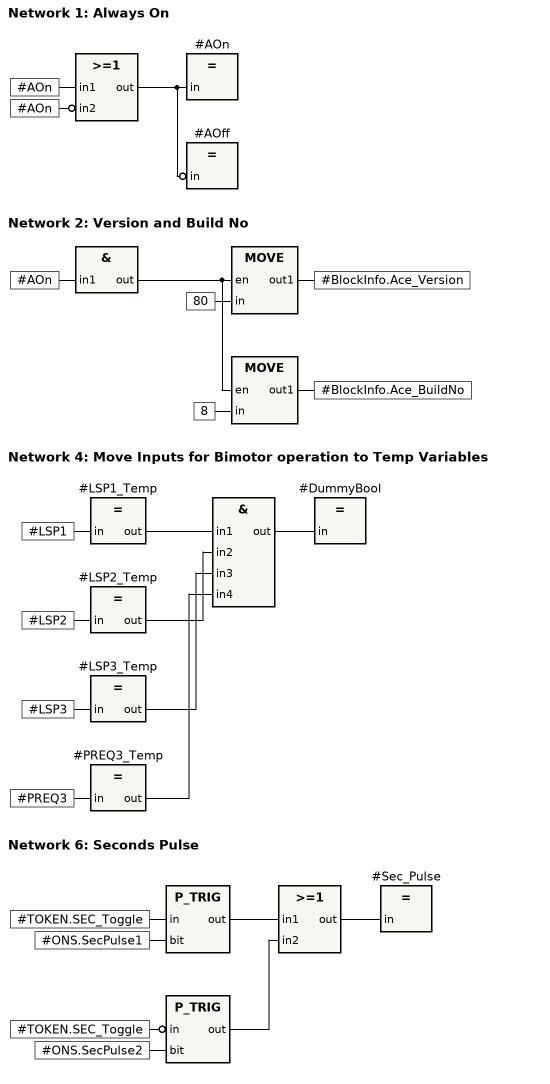
   #AOn := #AOn OR NOT #AOn;
   #AOff := NOT #AOn;
END_REGION

REGION Network 2: Version and Build No
   IF #AOn THEN
       #BlockInfo.Ace_Version := 80;
       #BlockInfo.Ace_BuildNo := 8;
   END_IF;
END_REGION

REGION Network 3 (STL): Instance DB Number to Faceplate
         L     DINO;
         T     #BlockInfo.DB_Number;
END_REGION

REGION Network 4: Move Inputs for Bimotor operation to Temp Variables
   #LSP1_Temp := #LSP1;
   #LSP2_Temp := #LSP2;
   #LSP3_Temp := #LSP3;
   #PREQ3_Temp := #PREQ3;
   #DummyBool := #LSP1 AND #LSP2 AND #LSP3 AND #PREQ3;
END_REGION

REGION Network 5 (SCL): Transfer Interlock OK to Stat
   #OUT.INTL_OK_STAT := PEEK_BOOL(area := 16#84, dbNumber := #BlockInfo.DB_Number, byteOffset := 18, bitOffset := 0);
   #OUT.INTL_SEQ_STR1_OK_STAT := PEEK_BOOL(area := 16#84, dbNumber := #BlockInfo.DB_Number, byteOffset := 20, bitOffset := 0);
   #OUT.INTL_SEQ_STR2_OK_STAT := PEEK_BOOL(area := 16#84, dbNumber := #BlockInfo.DB_Number, byteOffset := 22, bitOffset := 0);
   #OUT.INTL_SEQ_STR3_OK_STAT := PEEK_BOOL(area := 16#84, dbNumber := #BlockInfo.DB_Number, byteOffset := 24, bitOffset := 0);
   #OUT.INTL_SEQ_STP_OK_STAT := PEEK_BOOL(area := 16#84, dbNumber := #BlockInfo.DB_Number, byteOffset := 26, bitOffset := 0);
END_REGION

REGION Network 6: Seconds Pulse
   #_w1 := #TOKEN.SEC_Toggle AND NOT #ONS.SecPulse1;   // rising edge
   #ONS.SecPulse1 := #TOKEN.SEC_Toggle;
   #_w2 := NOT #TOKEN.SEC_Toggle AND NOT #ONS.SecPulse2;   // rising edge
   #ONS.SecPulse2 := NOT #TOKEN.SEC_Toggle;
   #Sec_Pulse := #_w1 OR #_w2;
END_REGION

REGION Network 7: Type Select
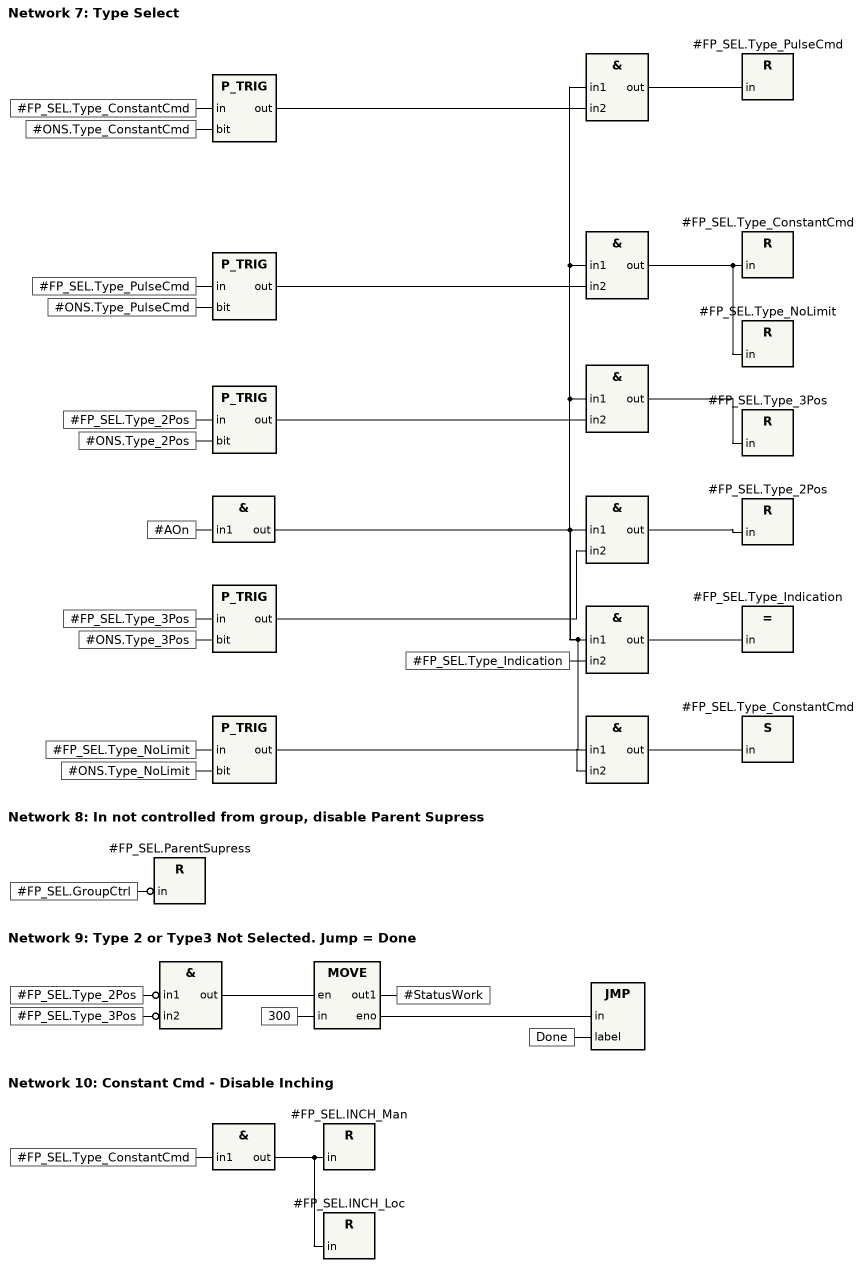
   #_w1 := #FP_SEL.Type_ConstantCmd AND NOT #ONS.Type_ConstantCmd;   // rising edge
   #ONS.Type_ConstantCmd := #FP_SEL.Type_ConstantCmd;
   IF #AOn AND #_w1 THEN #FP_SEL.Type_PulseCmd := FALSE; END_IF;
   #_w2 := #FP_SEL.Type_PulseCmd AND NOT #ONS.Type_PulseCmd;   // rising edge
   #ONS.Type_PulseCmd := #FP_SEL.Type_PulseCmd;
   IF #AOn AND #_w2 THEN
       #FP_SEL.Type_ConstantCmd := FALSE;
       #FP_SEL.Type_NoLimit := FALSE;
   END_IF;
   #_w3 := #FP_SEL.Type_2Pos AND NOT #ONS.Type_2Pos;   // rising edge
   #ONS.Type_2Pos := #FP_SEL.Type_2Pos;
   IF #AOn AND #_w3 THEN #FP_SEL.Type_3Pos := FALSE; END_IF;
   #_w4 := #FP_SEL.Type_3Pos AND NOT #ONS.Type_3Pos;   // rising edge
   #ONS.Type_3Pos := #FP_SEL.Type_3Pos;
   IF #AOn AND #_w4 THEN #FP_SEL.Type_2Pos := FALSE; END_IF;
   #FP_SEL.Type_Indication := #AOn AND #FP_SEL.Type_Indication;
   #_w5 := #FP_SEL.Type_NoLimit AND NOT #ONS.Type_NoLimit;   // rising edge
   #ONS.Type_NoLimit := #FP_SEL.Type_NoLimit;
   IF #AOn AND #_w5 THEN #FP_SEL.Type_ConstantCmd := TRUE; END_IF;
END_REGION

REGION Network 8: In not controlled from group, disable Parent Supress
   IF NOT #FP_SEL.GroupCtrl THEN #FP_SEL.ParentSupress := FALSE; END_IF;
END_REGION

REGION Network 9: Type 2 or Type3 Not Selected. Jump = Done
   // ENO of a box is taken as its EN; it also drops when the box reports an error
   #_w1 := NOT #FP_SEL.Type_2Pos AND NOT #FP_SEL.Type_3Pos;
   IF #_w1 THEN
       #StatusWork := 300;
       GOTO Done;
   END_IF;
END_REGION

REGION Network 10: Constant Cmd - Disable Inching
   IF #FP_SEL.Type_ConstantCmd THEN
       #FP_SEL.INCH_Man := FALSE;
       #FP_SEL.INCH_Loc := FALSE;
   END_IF;
END_REGION

REGION Network 11: Simulate LSP if no limit switches
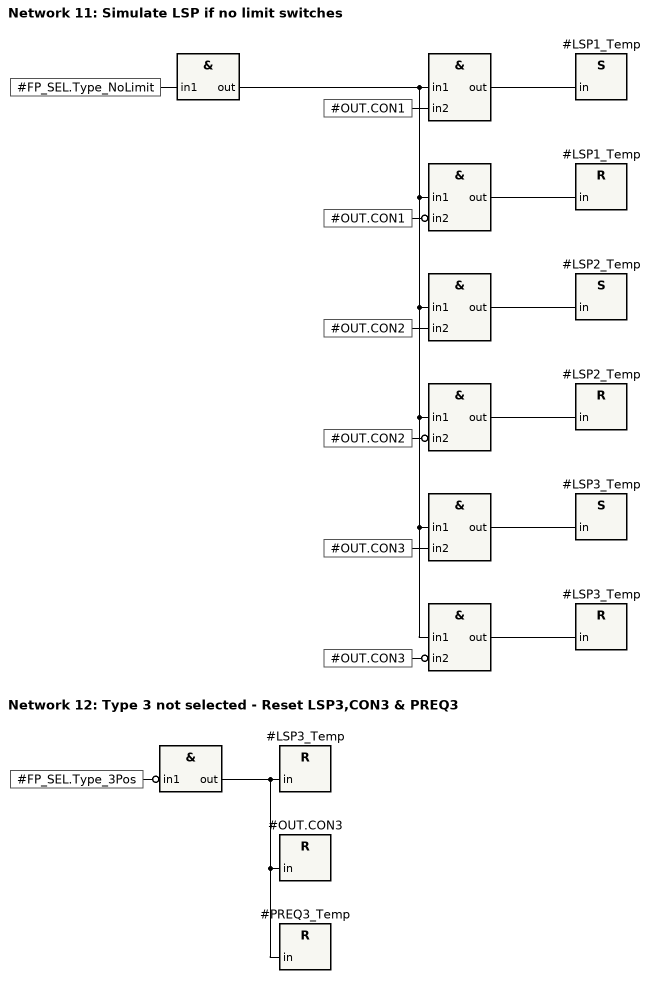
   IF #FP_SEL.Type_NoLimit AND #OUT.CON1 THEN #LSP1_Temp := TRUE; END_IF;
   IF #FP_SEL.Type_NoLimit AND NOT #OUT.CON1 THEN #LSP1_Temp := FALSE; END_IF;
   IF #FP_SEL.Type_NoLimit AND #OUT.CON2 THEN #LSP2_Temp := TRUE; END_IF;
   IF #FP_SEL.Type_NoLimit AND NOT #OUT.CON2 THEN #LSP2_Temp := FALSE; END_IF;
   IF #FP_SEL.Type_NoLimit AND #OUT.CON3 THEN #LSP3_Temp := TRUE; END_IF;
   IF #FP_SEL.Type_NoLimit AND NOT #OUT.CON3 THEN #LSP3_Temp := FALSE; END_IF;
END_REGION

REGION Network 12: Type 3 not selected - Reset LSP3,CON3 & PREQ3
   IF NOT #FP_SEL.Type_3Pos THEN
       #LSP3_Temp := FALSE;
       #OUT.CON3 := FALSE;
       #PREQ3_Temp := FALSE;
   END_IF;
END_REGION

REGION Network 13: Set Show Parameters
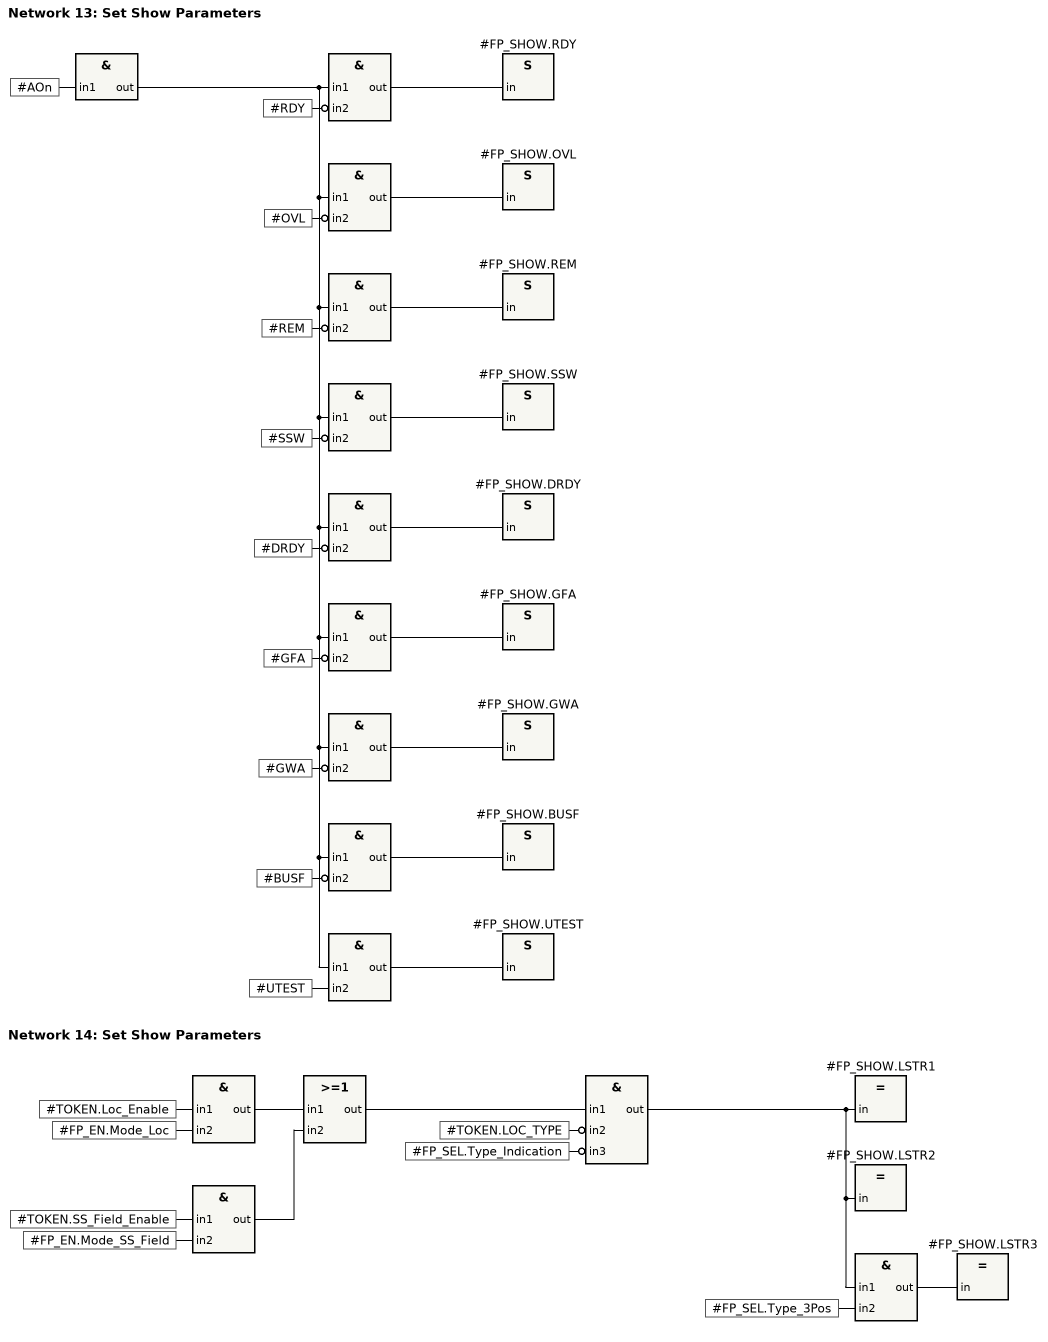
   IF #AOn AND NOT #RDY THEN #FP_SHOW.RDY := TRUE; END_IF;
   IF #AOn AND NOT #OVL THEN #FP_SHOW.OVL := TRUE; END_IF;
   IF #AOn AND NOT #REM THEN #FP_SHOW.REM := TRUE; END_IF;
   IF #AOn AND NOT #SSW THEN #FP_SHOW.SSW := TRUE; END_IF;
   IF #AOn AND NOT #DRDY THEN #FP_SHOW.DRDY := TRUE; END_IF;
   IF #AOn AND NOT #GFA THEN #FP_SHOW.GFA := TRUE; END_IF;
   IF #AOn AND NOT #GWA THEN #FP_SHOW.GWA := TRUE; END_IF;
   IF #AOn AND NOT #BUSF THEN #FP_SHOW.BUSF := TRUE; END_IF;
   IF #AOn AND #UTEST THEN #FP_SHOW.UTEST := TRUE; END_IF;
END_REGION

REGION Network 14: Set Show Parameters
   #FP_SHOW.LSTR1 := ((#TOKEN.Loc_Enable AND #FP_EN.Mode_Loc) OR (#TOKEN.SS_Field_Enable AND #FP_EN.Mode_SS_Field)) AND NOT #TOKEN.LOC_TYPE AND NOT #FP_SEL.Type_Indication;
   #FP_SHOW.LSTR2 := #FP_SHOW.LSTR1;
   #FP_SHOW.LSTR3 := #FP_SHOW.LSTR1 AND #FP_SEL.Type_3Pos;
END_REGION

REGION Network 15: Set Show Parameters
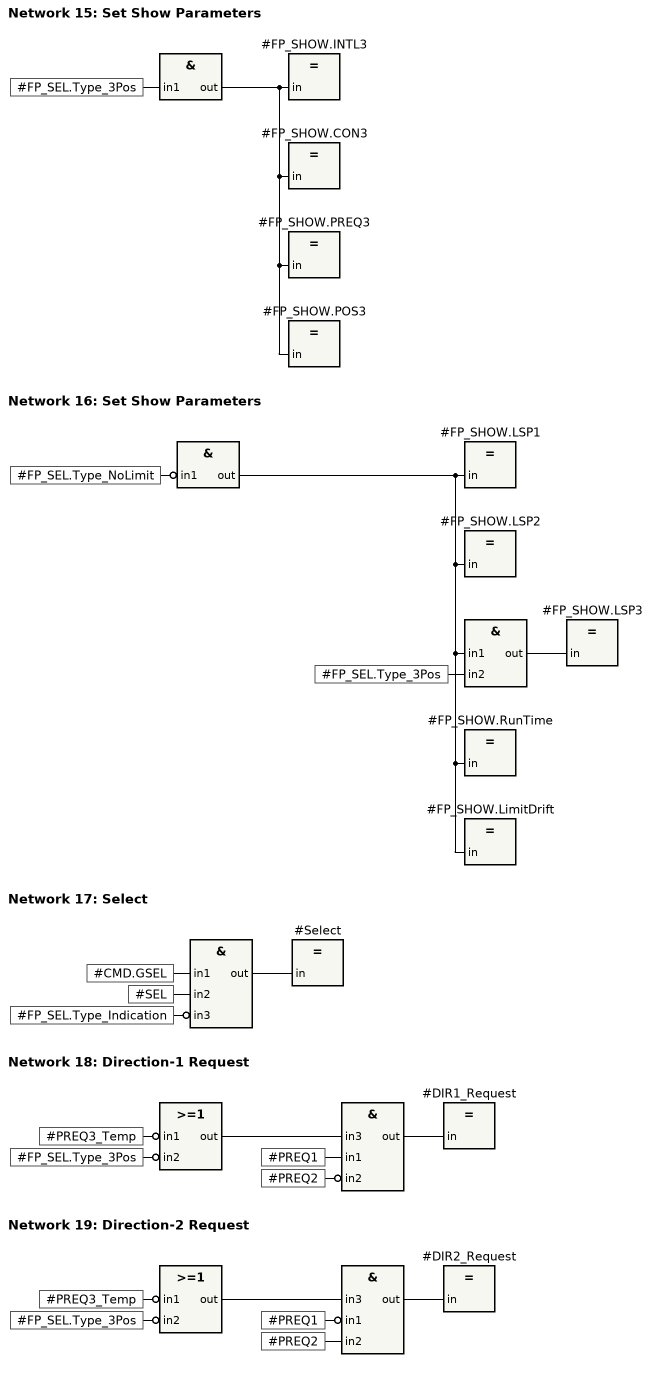
   #FP_SHOW.INTL3 := #FP_SEL.Type_3Pos;
   #FP_SHOW.CON3 := #FP_SEL.Type_3Pos;
   #FP_SHOW.PREQ3 := #FP_SEL.Type_3Pos;
   #FP_SHOW.POS3 := #FP_SEL.Type_3Pos;
END_REGION

REGION Network 16: Set Show Parameters
   #FP_SHOW.LSP1 := NOT #FP_SEL.Type_NoLimit;
   #FP_SHOW.LSP2 := NOT #FP_SEL.Type_NoLimit;
   #FP_SHOW.LSP3 := NOT #FP_SEL.Type_NoLimit AND #FP_SEL.Type_3Pos;
   #FP_SHOW.RunTime := NOT #FP_SEL.Type_NoLimit;
   #FP_SHOW.LimitDrift := NOT #FP_SEL.Type_NoLimit;
END_REGION

REGION Network 17: Select
   #Select := #CMD.GSEL AND #SEL AND NOT #FP_SEL.Type_Indication;
END_REGION

REGION Network 18: Direction-1 Request
   #DIR1_Request := (NOT #PREQ3_Temp OR NOT #FP_SEL.Type_3Pos) AND #PREQ1 AND NOT #PREQ2;
END_REGION

REGION Network 19: Direction-2 Request
   #DIR2_Request := (NOT #PREQ3_Temp OR NOT #FP_SEL.Type_3Pos) AND NOT #PREQ1 AND #PREQ2;
END_REGION

REGION Network 20: Direction-3 Request
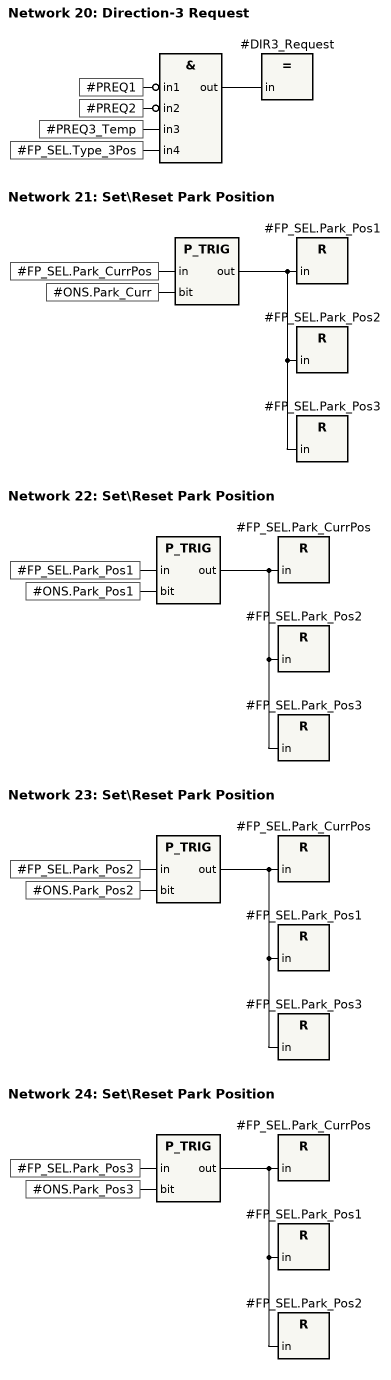
   #DIR3_Request := NOT #PREQ1 AND NOT #PREQ2 AND #PREQ3_Temp AND #FP_SEL.Type_3Pos;
END_REGION

REGION Network 21: Set\Reset Park Position
   #_w1 := #FP_SEL.Park_CurrPos AND NOT #ONS.Park_Curr;   // rising edge
   #ONS.Park_Curr := #FP_SEL.Park_CurrPos;
   IF #_w1 THEN
       #FP_SEL.Park_Pos1 := FALSE;
       #FP_SEL.Park_Pos2 := FALSE;
       #FP_SEL.Park_Pos3 := FALSE;
   END_IF;
END_REGION

REGION Network 22: Set\Reset Park Position
   #_w1 := #FP_SEL.Park_Pos1 AND NOT #ONS.Park_Pos1;   // rising edge
   #ONS.Park_Pos1 := #FP_SEL.Park_Pos1;
   IF #_w1 THEN
       #FP_SEL.Park_CurrPos := FALSE;
       #FP_SEL.Park_Pos2 := FALSE;
       #FP_SEL.Park_Pos3 := FALSE;
   END_IF;
END_REGION

REGION Network 23: Set\Reset Park Position
   #_w1 := #FP_SEL.Park_Pos2 AND NOT #ONS.Park_Pos2;   // rising edge
   #ONS.Park_Pos2 := #FP_SEL.Park_Pos2;
   IF #_w1 THEN
       #FP_SEL.Park_CurrPos := FALSE;
       #FP_SEL.Park_Pos1 := FALSE;
       #FP_SEL.Park_Pos3 := FALSE;
   END_IF;
END_REGION

REGION Network 24: Set\Reset Park Position
   #_w1 := #FP_SEL.Park_Pos3 AND NOT #ONS.Park_Pos3;   // rising edge
   #ONS.Park_Pos3 := #FP_SEL.Park_Pos3;
   IF #_w1 THEN
       #FP_SEL.Park_CurrPos := FALSE;
       #FP_SEL.Park_Pos1 := FALSE;
       #FP_SEL.Park_Pos2 := FALSE;
   END_IF;
END_REGION

REGION Network 25: Set\Reset Park Position
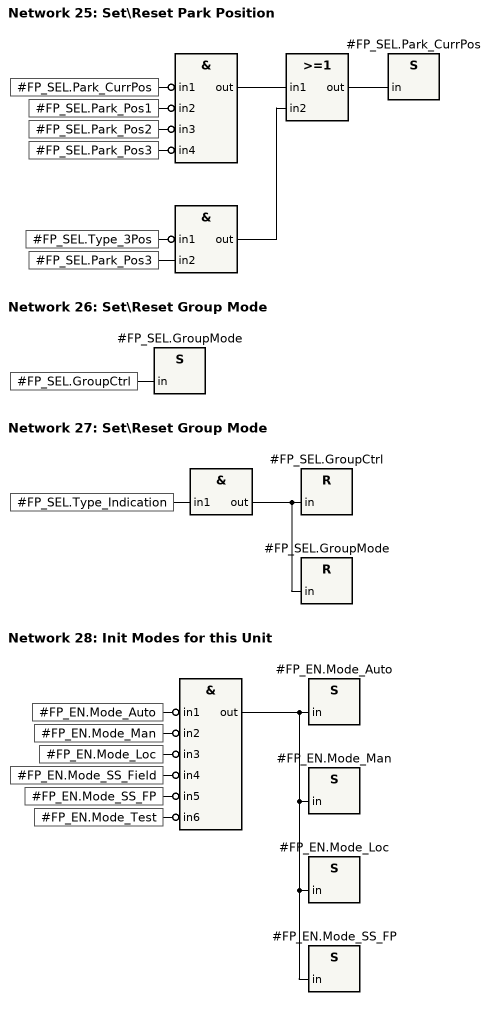
   IF (NOT #FP_SEL.Park_CurrPos AND NOT #FP_SEL.Park_Pos1 AND NOT #FP_SEL.Park_Pos2 AND NOT #FP_SEL.Park_Pos3) OR (NOT #FP_SEL.Type_3Pos AND #FP_SEL.Park_Pos3) THEN
       #FP_SEL.Park_CurrPos := TRUE;
   END_IF;
END_REGION

REGION Network 26: Set\Reset Group Mode
   IF #FP_SEL.GroupCtrl THEN #FP_SEL.GroupMode := TRUE; END_IF;
END_REGION

REGION Network 27: Set\Reset Group Mode
   IF #FP_SEL.Type_Indication THEN
       #FP_SEL.GroupCtrl := FALSE;
       #FP_SEL.GroupMode := FALSE;
   END_IF;
END_REGION

REGION Network 28: Init Modes for this Unit
   #_w1 := NOT #FP_EN.Mode_Auto AND NOT #FP_EN.Mode_Man AND NOT #FP_EN.Mode_Loc AND NOT #FP_EN.Mode_SS_Field AND NOT #FP_EN.Mode_SS_FP AND NOT #FP_EN.Mode_Test;
   IF #_w1 THEN
       #FP_EN.Mode_Auto := TRUE;
       #FP_EN.Mode_Man := TRUE;
       #FP_EN.Mode_Loc := TRUE;
       #FP_EN.Mode_SS_FP := TRUE;
   END_IF;
END_REGION

REGION Network 29: Show Push Buttons on Faceplate
   // build 002 - 27 March 2019 : LOC_Type flag removed from Show_PB_Local
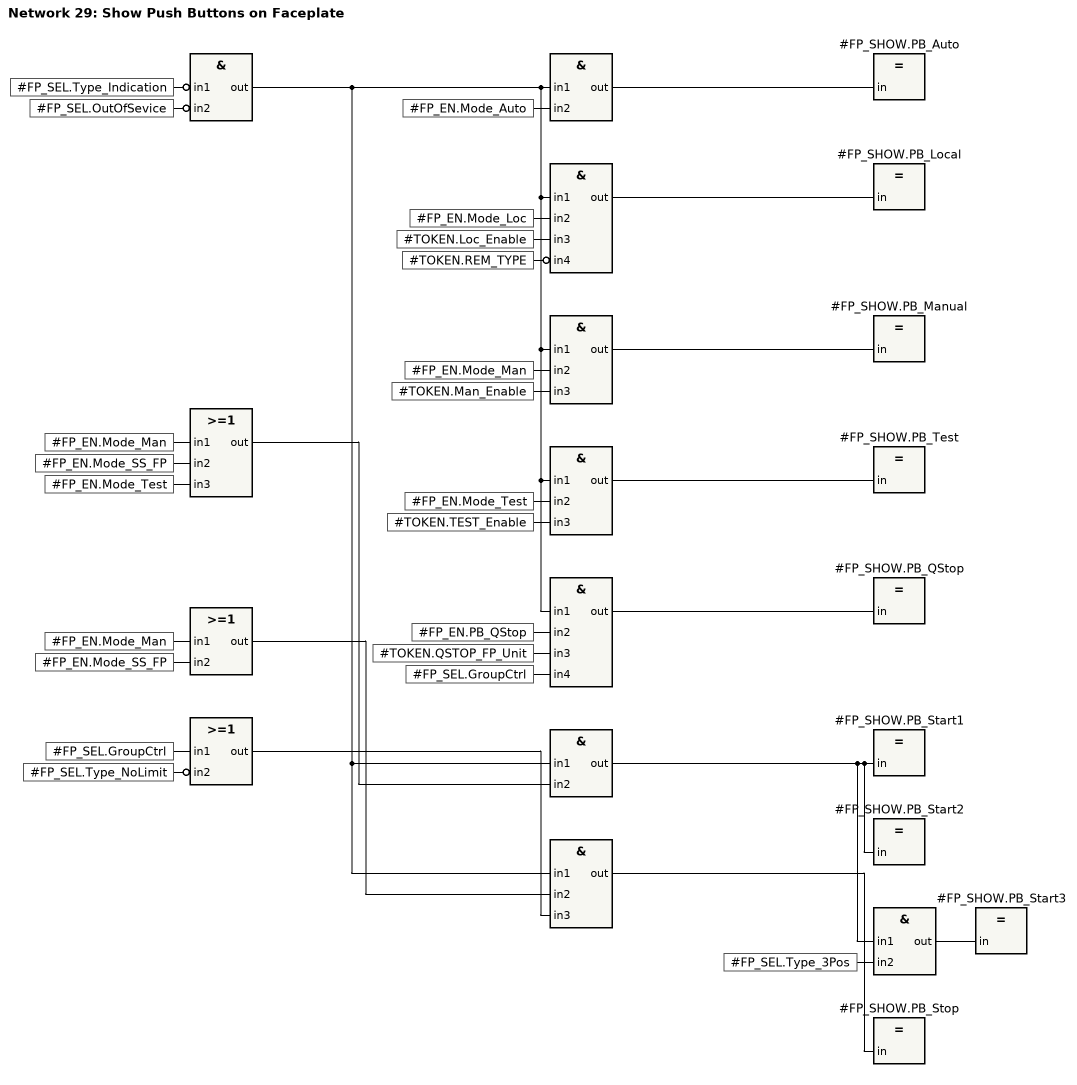
   #_w1 := NOT #FP_SEL.Type_Indication AND NOT #FP_SEL.OutOfSevice;
   #FP_SHOW.PB_Auto := #_w1 AND #FP_EN.Mode_Auto;
   #FP_SHOW.PB_Local := #_w1 AND #FP_EN.Mode_Loc AND #TOKEN.Loc_Enable AND NOT #TOKEN.REM_TYPE;
   #FP_SHOW.PB_Manual := #_w1 AND #FP_EN.Mode_Man AND #TOKEN.Man_Enable;
   #FP_SHOW.PB_Test := #_w1 AND #FP_EN.Mode_Test AND #TOKEN.TEST_Enable;
   #FP_SHOW.PB_QStop := #_w1 AND #FP_EN.PB_QStop AND #TOKEN.QSTOP_FP_Unit AND #FP_SEL.GroupCtrl;
   #FP_SHOW.PB_Start1 := #_w1 AND (#FP_EN.Mode_Man OR #FP_EN.Mode_SS_FP OR #FP_EN.Mode_Test);
   #FP_SHOW.PB_Start2 := #FP_SHOW.PB_Start1;
   #FP_SHOW.PB_Start3 := #FP_SHOW.PB_Start1 AND #FP_SEL.Type_3Pos;
   #FP_SHOW.PB_Stop := #_w1 AND (#FP_EN.Mode_Man OR #FP_EN.Mode_SS_FP) AND (#FP_SEL.GroupCtrl OR NOT #FP_SEL.Type_NoLimit);
END_REGION

REGION Network 30: DimOut Buttons on Faceplate - Auto
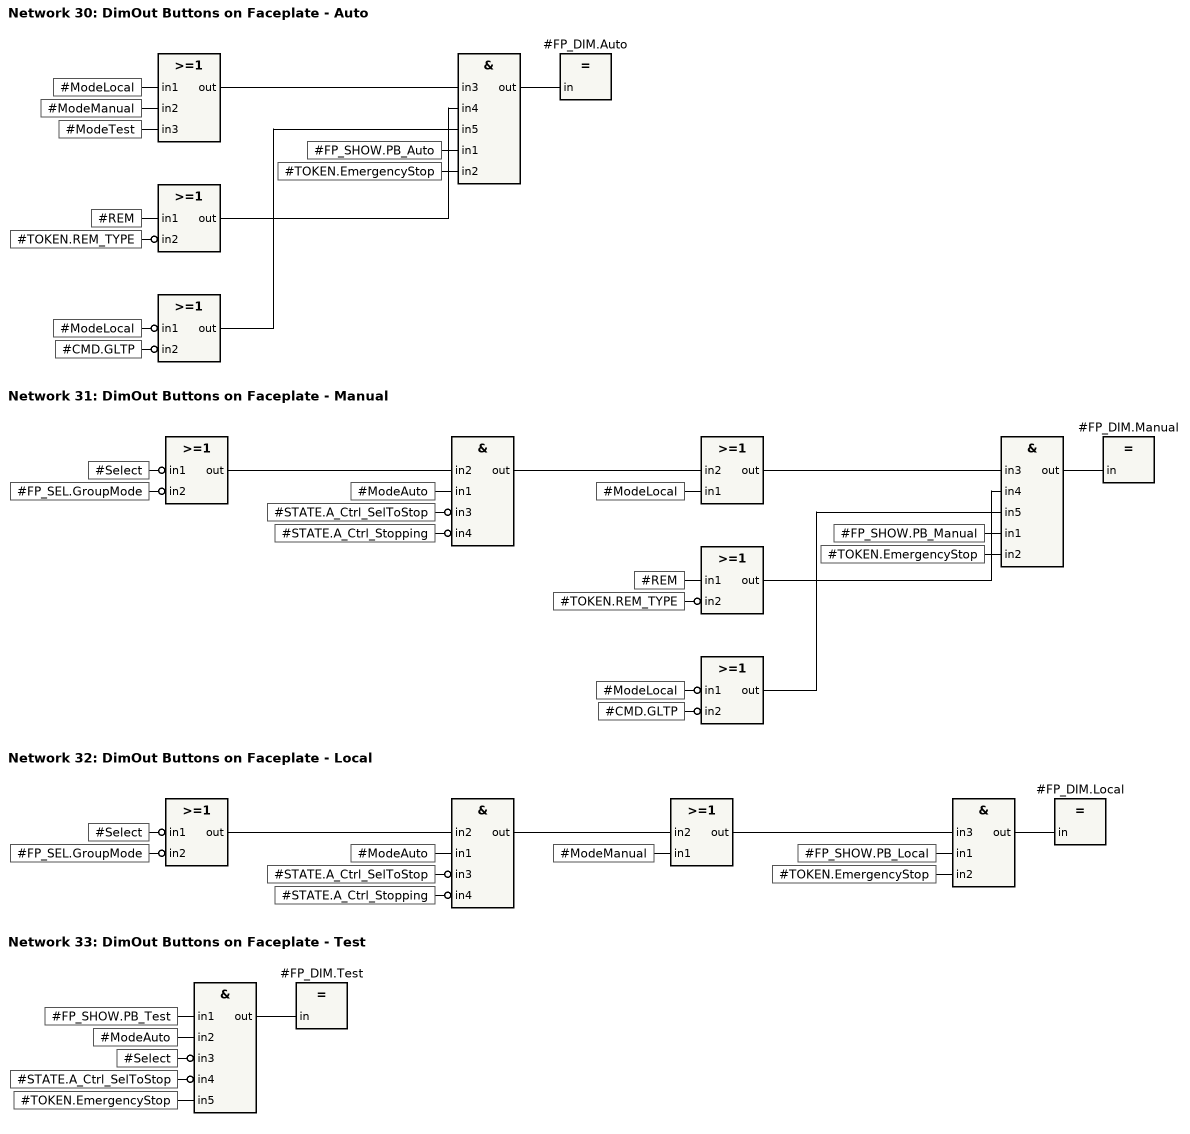
   #FP_DIM.Auto := (#ModeLocal OR #ModeManual OR #ModeTest) AND (#REM OR NOT #TOKEN.REM_TYPE) AND (NOT #ModeLocal OR NOT #CMD.GLTP) AND #FP_SHOW.PB_Auto AND #TOKEN.EmergencyStop;
END_REGION

REGION Network 31: DimOut Buttons on Faceplate - Manual
   #FP_DIM.Manual := (((NOT #Select OR NOT #FP_SEL.GroupMode) AND #ModeAuto AND NOT #STATE.A_Ctrl_SelToStop AND NOT #STATE.A_Ctrl_Stopping) OR #ModeLocal) AND (#REM OR NOT #TOKEN.REM_TYPE) AND (NOT #ModeLocal OR NOT #CMD.GLTP) AND #FP_SHOW.PB_Manual AND #TOKEN.EmergencyStop;
END_REGION

REGION Network 32: DimOut Buttons on Faceplate - Local
   #FP_DIM.Local := (((NOT #Select OR NOT #FP_SEL.GroupMode) AND #ModeAuto AND NOT #STATE.A_Ctrl_SelToStop AND NOT #STATE.A_Ctrl_Stopping) OR #ModeManual) AND #FP_SHOW.PB_Local AND #TOKEN.EmergencyStop;
END_REGION

REGION Network 33: DimOut Buttons on Faceplate - Test
   #FP_DIM.Test := #FP_SHOW.PB_Test AND #ModeAuto AND NOT #Select AND NOT #STATE.A_Ctrl_SelToStop AND #TOKEN.EmergencyStop;
END_REGION

REGION Network 34: DimOut Buttons on Faceplate - Stop
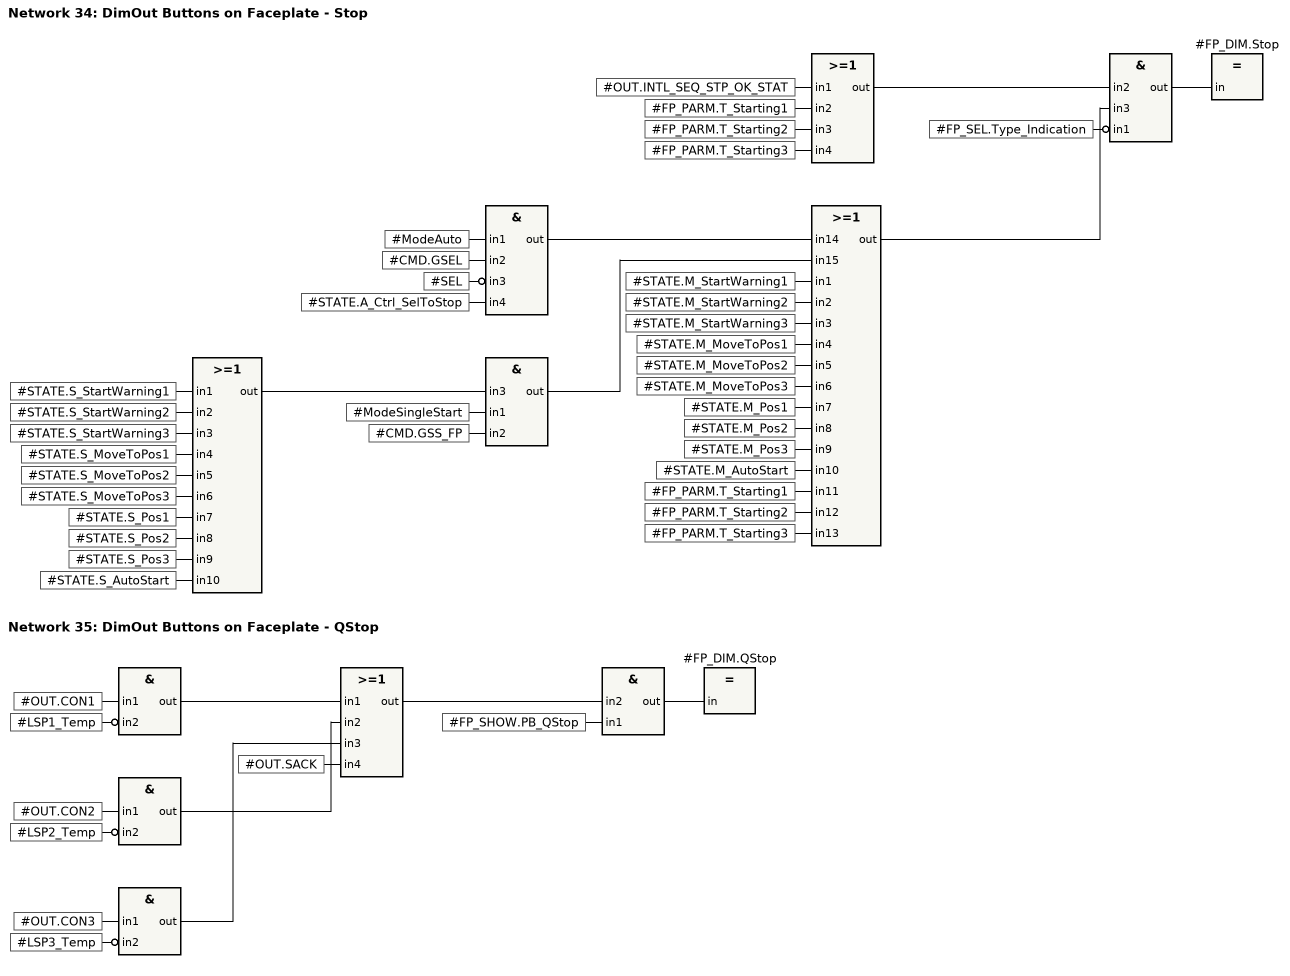
   #FP_DIM.Stop := (#OUT.INTL_SEQ_STP_OK_STAT OR #FP_PARM.T_Starting1 OR #FP_PARM.T_Starting2 OR #FP_PARM.T_Starting3) AND ((#ModeAuto AND #CMD.GSEL AND NOT #SEL AND #STATE.A_Ctrl_SelToStop) OR ((#STATE.S_StartWarning1 OR #STATE.S_StartWarning2 OR #STATE.S_StartWarning3 OR #STATE.S_MoveToPos1 OR #STATE.S_MoveToPos2 OR #STATE.S_MoveToPos3 OR #STATE.S_Pos1 OR #STATE.S_Pos2 OR #STATE.S_Pos3 OR #STATE.S_AutoStart) AND #ModeSingleStart AND #CMD.GSS_FP) OR #STATE.M_StartWarning1 OR #STATE.M_StartWarning2 OR #STATE.M_StartWarning3 OR #STATE.M_MoveToPos1 OR #STATE.M_MoveToPos2 OR #STATE.M_MoveToPos3 OR #STATE.M_Pos1 OR #STATE.M_Pos2 OR #STATE.M_Pos3 OR #STATE.M_AutoStart OR #FP_PARM.T_Starting1 OR #FP_PARM.T_Starting2 OR #FP_PARM.T_Starting3) AND NOT #FP_SEL.Type_Indication;
END_REGION

REGION Network 35: DimOut Buttons on Faceplate - QStop
   #FP_DIM.QStop := ((#OUT.CON1 AND NOT #LSP1_Temp) OR (#OUT.CON2 AND NOT #LSP2_Temp) OR (#OUT.CON3 AND NOT #LSP3_Temp) OR #OUT.SACK) AND #FP_SHOW.PB_QStop;
END_REGION

REGION Network 36: DimOut Buttons on Faceplate - Start1
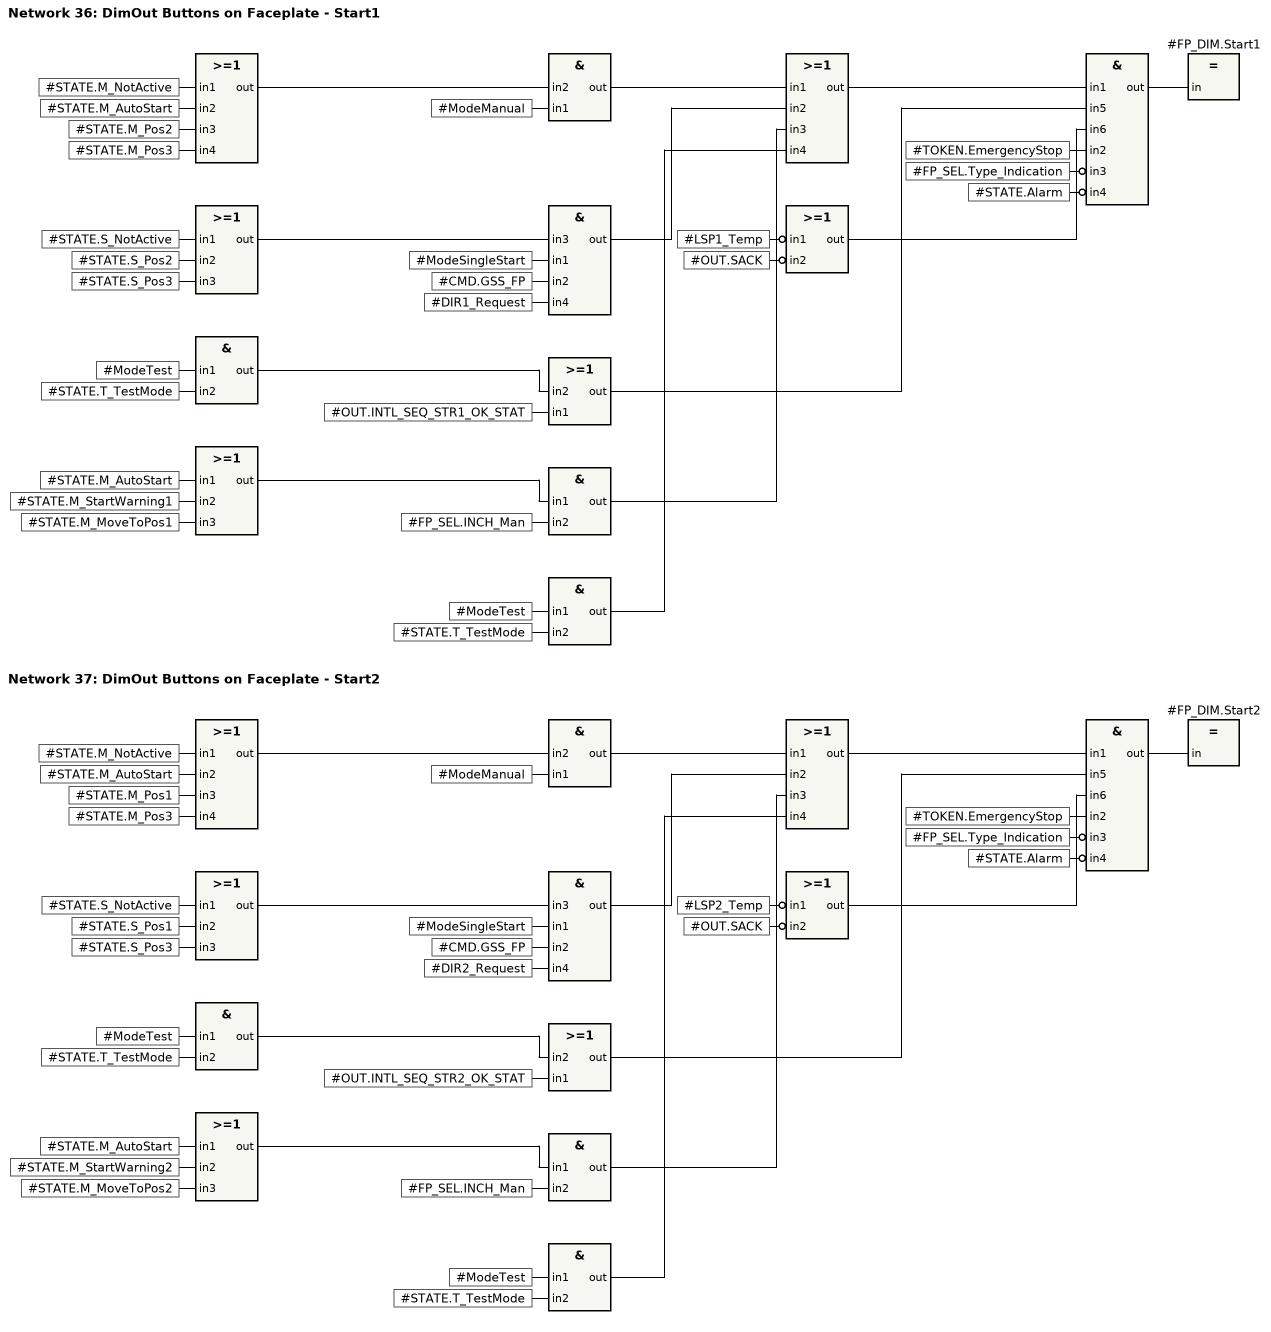
   #FP_DIM.Start1 := (((#STATE.M_NotActive OR #STATE.M_AutoStart OR #STATE.M_Pos2 OR #STATE.M_Pos3) AND #ModeManual) OR ((#STATE.S_NotActive OR #STATE.S_Pos2 OR #STATE.S_Pos3) AND #ModeSingleStart AND #CMD.GSS_FP AND #DIR1_Request) OR ((#STATE.M_AutoStart OR #STATE.M_StartWarning1 OR #STATE.M_MoveToPos1) AND #FP_SEL.INCH_Man) OR (#ModeTest AND #STATE.T_TestMode)) AND ((#ModeTest AND #STATE.T_TestMode) OR #OUT.INTL_SEQ_STR1_OK_STAT) AND (NOT #LSP1_Temp OR NOT #OUT.SACK) AND #TOKEN.EmergencyStop AND NOT #FP_SEL.Type_Indication AND NOT #STATE.Alarm;
END_REGION

REGION Network 37: DimOut Buttons on Faceplate - Start2
   #FP_DIM.Start2 := (((#STATE.M_NotActive OR #STATE.M_AutoStart OR #STATE.M_Pos1 OR #STATE.M_Pos3) AND #ModeManual) OR ((#STATE.S_NotActive OR #STATE.S_Pos1 OR #STATE.S_Pos3) AND #ModeSingleStart AND #CMD.GSS_FP AND #DIR2_Request) OR ((#STATE.M_AutoStart OR #STATE.M_StartWarning2 OR #STATE.M_MoveToPos2) AND #FP_SEL.INCH_Man) OR (#ModeTest AND #STATE.T_TestMode)) AND ((#ModeTest AND #STATE.T_TestMode) OR #OUT.INTL_SEQ_STR2_OK_STAT) AND (NOT #LSP2_Temp OR NOT #OUT.SACK) AND #TOKEN.EmergencyStop AND NOT #FP_SEL.Type_Indication AND NOT #STATE.Alarm;
END_REGION

REGION Network 38: DimOut Buttons on Faceplate - Start3
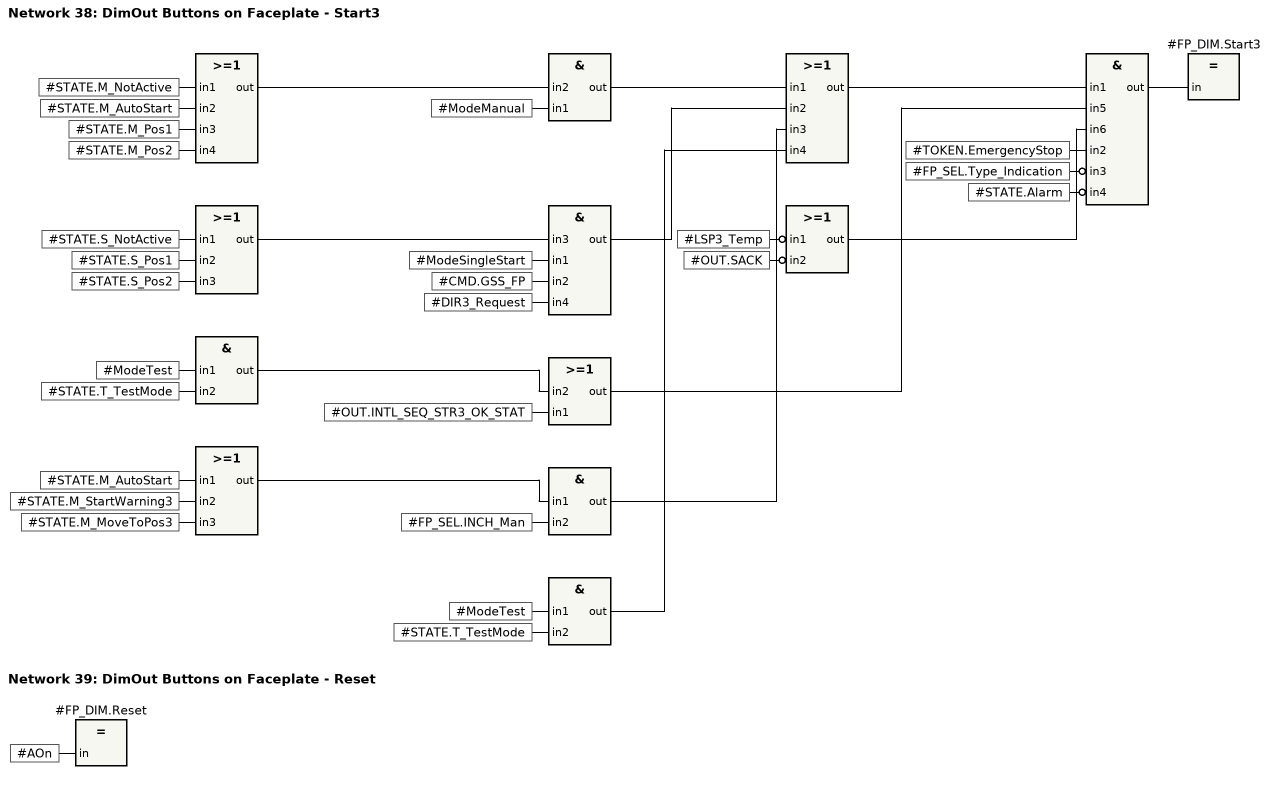
   #FP_DIM.Start3 := (((#STATE.M_NotActive OR #STATE.M_AutoStart OR #STATE.M_Pos1 OR #STATE.M_Pos2) AND #ModeManual) OR ((#STATE.S_NotActive OR #STATE.S_Pos1 OR #STATE.S_Pos2) AND #ModeSingleStart AND #CMD.GSS_FP AND #DIR3_Request) OR ((#STATE.M_AutoStart OR #STATE.M_StartWarning3 OR #STATE.M_MoveToPos3) AND #FP_SEL.INCH_Man) OR (#ModeTest AND #STATE.T_TestMode)) AND ((#ModeTest AND #STATE.T_TestMode) OR #OUT.INTL_SEQ_STR3_OK_STAT) AND (NOT #LSP3_Temp OR NOT #OUT.SACK) AND #TOKEN.EmergencyStop AND NOT #FP_SEL.Type_Indication AND NOT #STATE.Alarm;
END_REGION

REGION Network 39: DimOut Buttons on Faceplate - Reset
   #FP_DIM.Reset := #AOn;
END_REGION

REGION Network 40: MODE Handling - Auto Mode
   // Build 002 - 27 March 2019: REM flag is removed in FP_CMD.Auto commmand
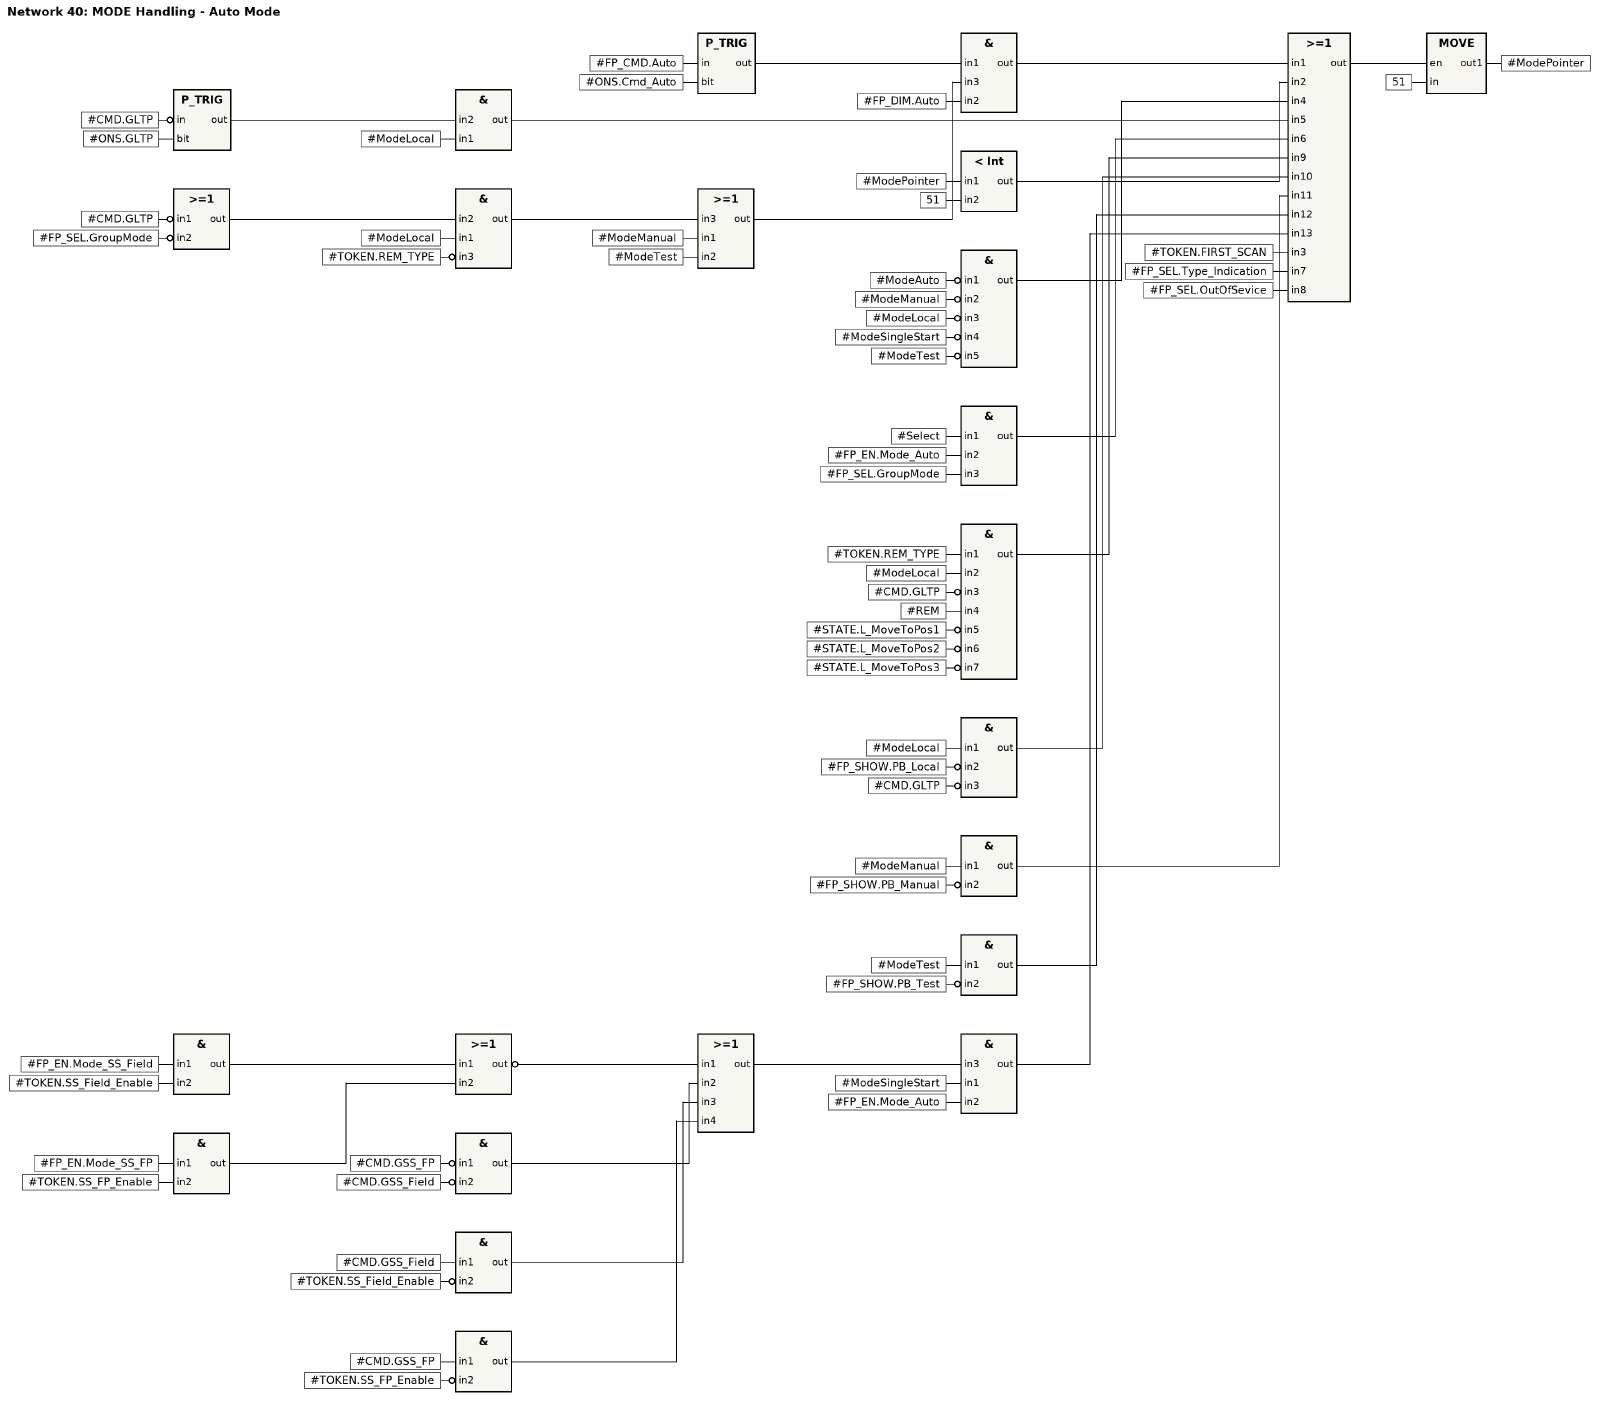
   #_w1 := #FP_CMD.Auto AND NOT #ONS.Cmd_Auto;   // rising edge
   #ONS.Cmd_Auto := #FP_CMD.Auto;
   #_w2 := NOT #CMD.GLTP AND NOT #ONS.GLTP;   // rising edge
   #ONS.GLTP := NOT #CMD.GLTP;
   IF (#_w1 AND (((NOT #CMD.GLTP OR NOT #FP_SEL.GroupMode) AND #ModeLocal AND NOT #TOKEN.REM_TYPE) OR #ModeManual OR #ModeTest) AND #FP_DIM.Auto) OR (#ModePointer < 51) OR (NOT #ModeAuto AND NOT #ModeManual AND NOT #ModeLocal AND NOT #ModeSingleStart AND NOT #ModeTest) OR (#_w2 AND #ModeLocal) OR (#Select AND #FP_EN.Mode_Auto AND #FP_SEL.GroupMode) OR (#TOKEN.REM_TYPE AND #ModeLocal AND NOT #CMD.GLTP AND #REM AND NOT #STATE.L_MoveToPos1 AND NOT #STATE.L_MoveToPos2 AND NOT #STATE.L_MoveToPos3) OR (#ModeLocal AND NOT #FP_SHOW.PB_Local AND NOT #CMD.GLTP) OR (#ModeManual AND NOT #FP_SHOW.PB_Manual) OR (#ModeTest AND NOT #FP_SHOW.PB_Test) OR ((NOT ((#FP_EN.Mode_SS_Field AND #TOKEN.SS_Field_Enable) OR (#FP_EN.Mode_SS_FP AND #TOKEN.SS_FP_Enable)) OR (NOT #CMD.GSS_FP AND NOT #CMD.GSS_Field) OR (#CMD.GSS_Field AND NOT #TOKEN.SS_Field_Enable) OR (#CMD.GSS_FP AND NOT #TOKEN.SS_FP_Enable)) AND #ModeSingleStart AND #FP_EN.Mode_Auto) OR #TOKEN.FIRST_SCAN OR #FP_SEL.Type_Indication OR #FP_SEL.OutOfSevice THEN
       #ModePointer := 51;
   END_IF;
END_REGION

REGION Network 41: MODE Handling - Manual Mode
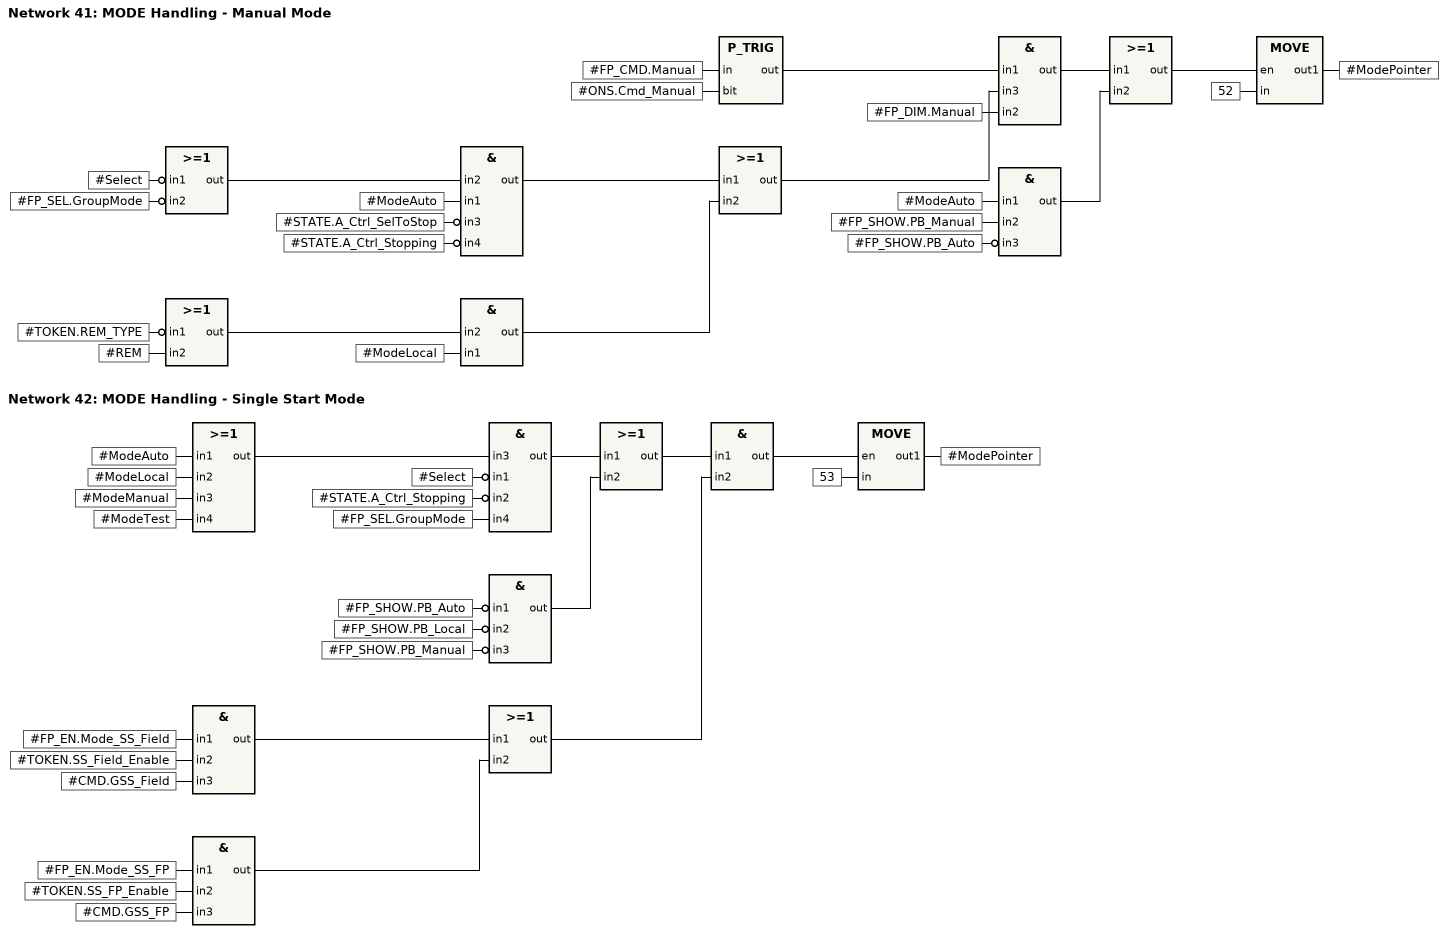
   #_w1 := #FP_CMD.Manual AND NOT #ONS.Cmd_Manual;   // rising edge
   #ONS.Cmd_Manual := #FP_CMD.Manual;
   IF (#_w1 AND (((NOT #Select OR NOT #FP_SEL.GroupMode) AND #ModeAuto AND NOT #STATE.A_Ctrl_SelToStop AND NOT #STATE.A_Ctrl_Stopping) OR ((NOT #TOKEN.REM_TYPE OR #REM) AND #ModeLocal)) AND #FP_DIM.Manual) OR (#ModeAuto AND #FP_SHOW.PB_Manual AND NOT #FP_SHOW.PB_Auto) THEN
       #ModePointer := 52;
   END_IF;
END_REGION

REGION Network 42: MODE Handling - Single Start Mode
   IF (((#ModeAuto OR #ModeLocal OR #ModeManual OR #ModeTest) AND NOT #Select AND NOT #STATE.A_Ctrl_Stopping AND #FP_SEL.GroupMode) OR (NOT #FP_SHOW.PB_Auto AND NOT #FP_SHOW.PB_Local AND NOT #FP_SHOW.PB_Manual)) AND ((#FP_EN.Mode_SS_Field AND #TOKEN.SS_Field_Enable AND #CMD.GSS_Field) OR (#FP_EN.Mode_SS_FP AND #TOKEN.SS_FP_Enable AND #CMD.GSS_FP)) THEN
       #ModePointer := 53;
   END_IF;
END_REGION

REGION Network 43: MODE Handling - Local Mode
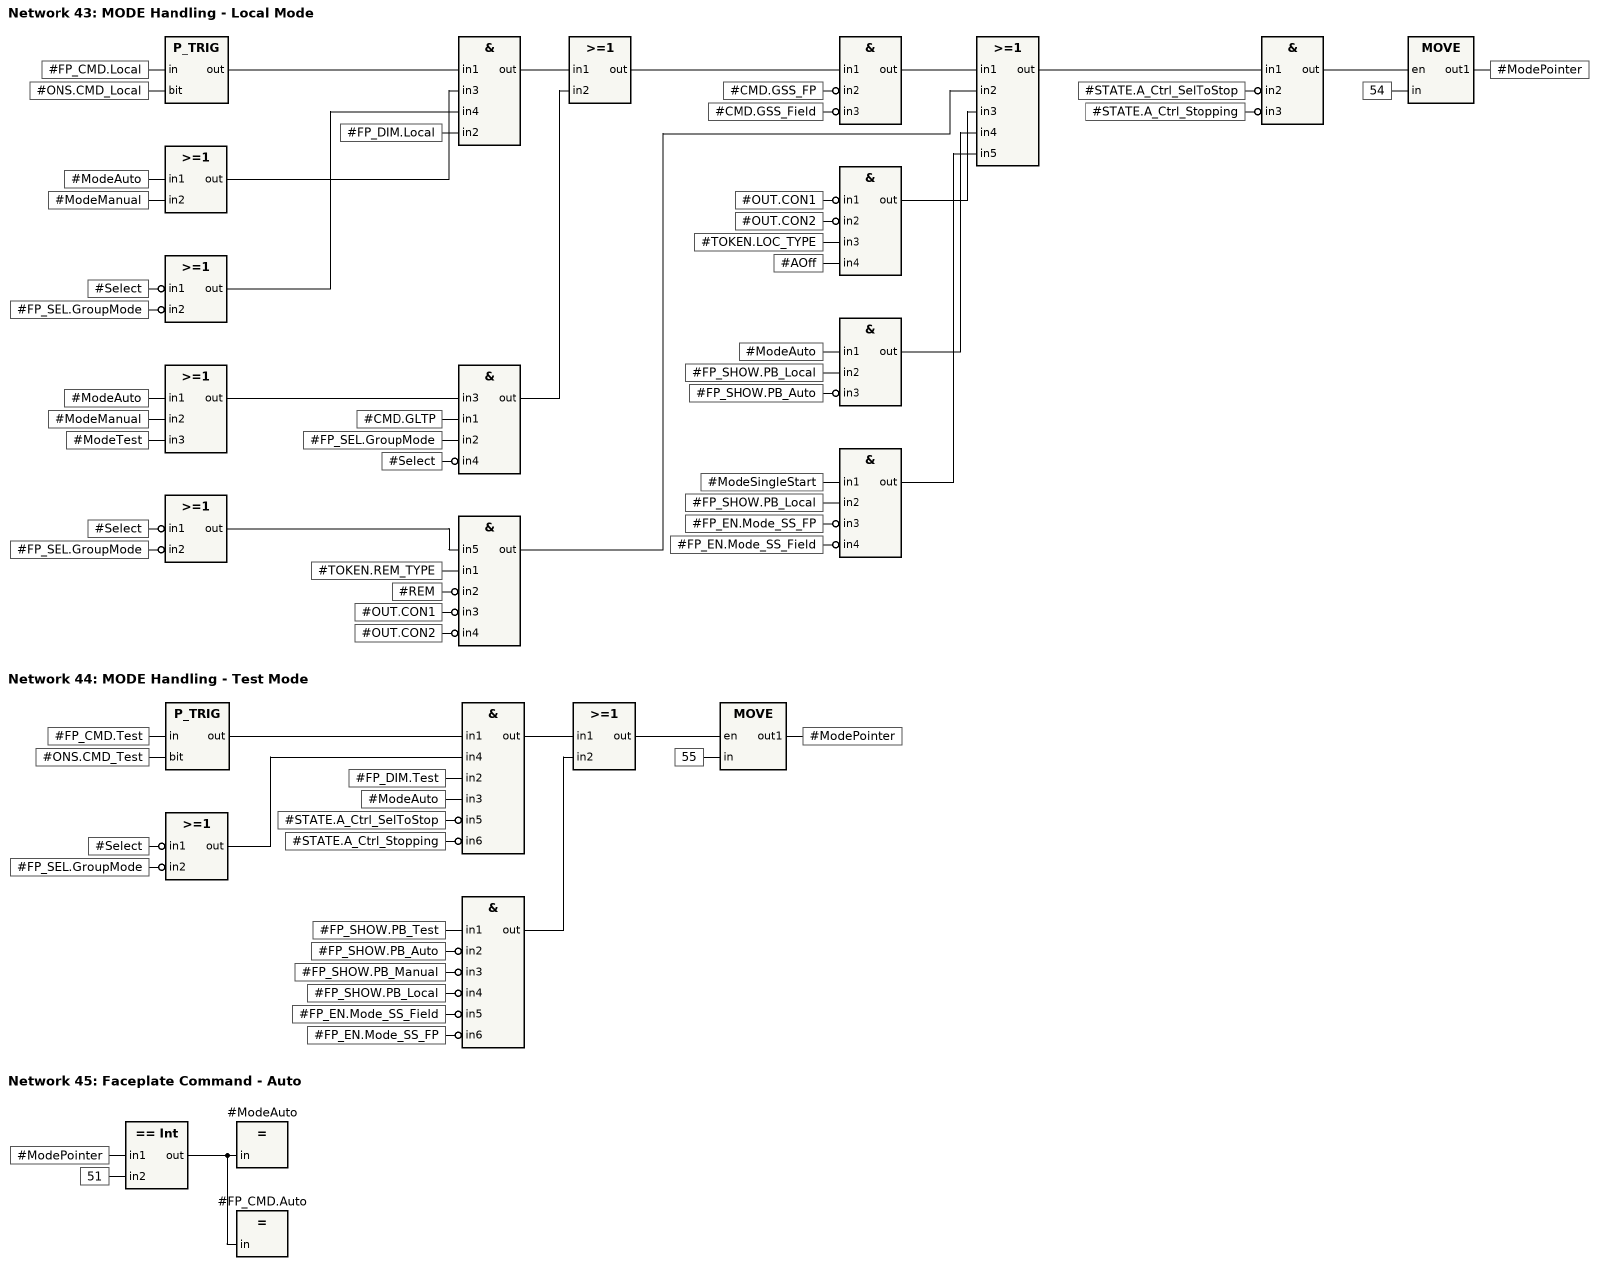
   #_w1 := #FP_CMD.Local AND NOT #ONS.CMD_Local;   // rising edge
   #ONS.CMD_Local := #FP_CMD.Local;
   IF ((((#_w1 AND (#ModeAuto OR #ModeManual) AND (NOT #Select OR NOT #FP_SEL.GroupMode) AND #FP_DIM.Local) OR ((#ModeAuto OR #ModeManual OR #ModeTest) AND #CMD.GLTP AND #FP_SEL.GroupMode AND NOT #Select)) AND NOT #CMD.GSS_FP AND NOT #CMD.GSS_Field) OR ((NOT #Select OR NOT #FP_SEL.GroupMode) AND #TOKEN.REM_TYPE AND NOT #REM AND NOT #OUT.CON1 AND NOT #OUT.CON2) OR (NOT #OUT.CON1 AND NOT #OUT.CON2 AND #TOKEN.LOC_TYPE AND #AOff) OR (#ModeAuto AND #FP_SHOW.PB_Local AND NOT #FP_SHOW.PB_Auto) OR (#ModeSingleStart AND #FP_SHOW.PB_Local AND NOT #FP_EN.Mode_SS_FP AND NOT #FP_EN.Mode_SS_Field)) AND NOT #STATE.A_Ctrl_SelToStop AND NOT #STATE.A_Ctrl_Stopping THEN
       #ModePointer := 54;
   END_IF;
END_REGION

REGION Network 44: MODE Handling - Test Mode
   #_w1 := #FP_CMD.Test AND NOT #ONS.CMD_Test;   // rising edge
   #ONS.CMD_Test := #FP_CMD.Test;
   IF (#_w1 AND (NOT #Select OR NOT #FP_SEL.GroupMode) AND #FP_DIM.Test AND #ModeAuto AND NOT #STATE.A_Ctrl_SelToStop AND NOT #STATE.A_Ctrl_Stopping) OR (#FP_SHOW.PB_Test AND NOT #FP_SHOW.PB_Auto AND NOT #FP_SHOW.PB_Manual AND NOT #FP_SHOW.PB_Local AND NOT #FP_EN.Mode_SS_Field AND NOT #FP_EN.Mode_SS_FP) THEN
       #ModePointer := 55;
   END_IF;
END_REGION

REGION Network 45: Faceplate Command - Auto
   #ModeAuto := #ModePointer = 51;
   #FP_CMD.Auto := #ModeAuto;
END_REGION

REGION Network 46: Faceplate Command - Manual
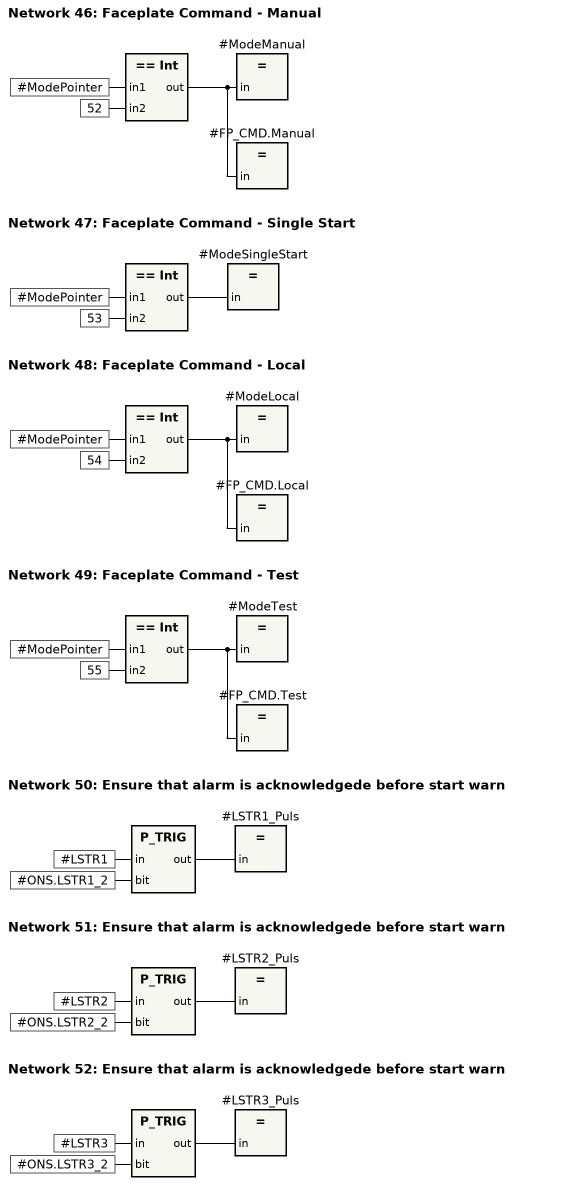
   #ModeManual := #ModePointer = 52;
   #FP_CMD.Manual := #ModeManual;
END_REGION

REGION Network 47: Faceplate Command - Single Start
   #ModeSingleStart := #ModePointer = 53;
END_REGION

REGION Network 48: Faceplate Command - Local
   #ModeLocal := #ModePointer = 54;
   #FP_CMD.Local := #ModeLocal;
END_REGION

REGION Network 49: Faceplate Command - Test
   #ModeTest := #ModePointer = 55;
   #FP_CMD.Test := #ModeTest;
END_REGION

REGION Network 50: Ensure that alarm is acknowledgede before start warn
   #_w1 := #LSTR1 AND NOT #ONS.LSTR1_2;   // rising edge
   #ONS.LSTR1_2 := #LSTR1;
   #LSTR1_Puls := #_w1;
END_REGION

REGION Network 51: Ensure that alarm is acknowledgede before start warn
   #_w1 := #LSTR2 AND NOT #ONS.LSTR2_2;   // rising edge
   #ONS.LSTR2_2 := #LSTR2;
   #LSTR2_Puls := #_w1;
END_REGION

REGION Network 52: Ensure that alarm is acknowledgede before start warn
   #_w1 := #LSTR3 AND NOT #ONS.LSTR3_2;   // rising edge
   #ONS.LSTR3_2 := #LSTR3;
   #LSTR3_Puls := #_w1;
END_REGION

REGION Network 53: Faceplate Commands Pulse Type - Start1
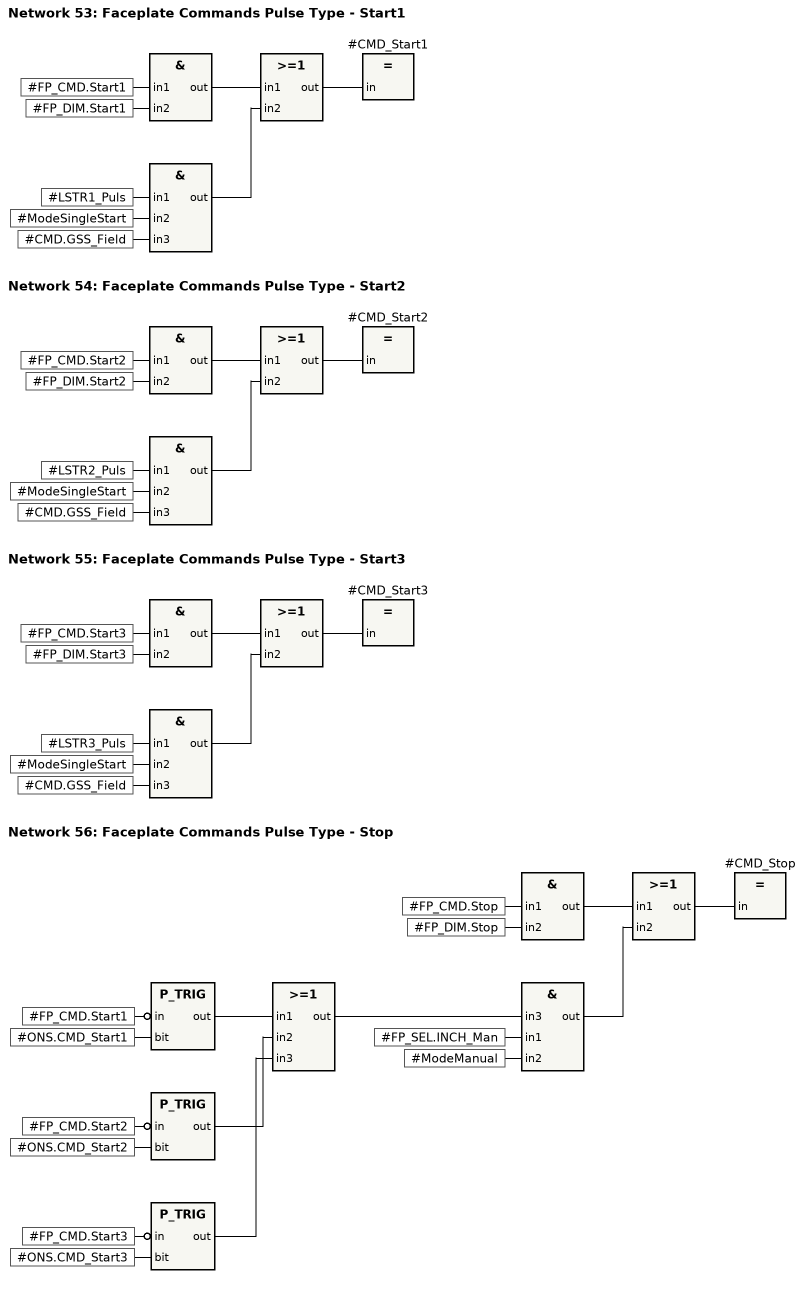
   #CMD_Start1 := (#FP_CMD.Start1 AND #FP_DIM.Start1) OR (#LSTR1_Puls AND #ModeSingleStart AND #CMD.GSS_Field);
END_REGION

REGION Network 54: Faceplate Commands Pulse Type - Start2
   #CMD_Start2 := (#FP_CMD.Start2 AND #FP_DIM.Start2) OR (#LSTR2_Puls AND #ModeSingleStart AND #CMD.GSS_Field);
END_REGION

REGION Network 55: Faceplate Commands Pulse Type - Start3
   #CMD_Start3 := (#FP_CMD.Start3 AND #FP_DIM.Start3) OR (#LSTR3_Puls AND #ModeSingleStart AND #CMD.GSS_Field);
END_REGION

REGION Network 56: Faceplate Commands Pulse Type - Stop
   #_w1 := NOT #FP_CMD.Start1 AND NOT #ONS.CMD_Start1;   // rising edge
   #ONS.CMD_Start1 := NOT #FP_CMD.Start1;
   #_w2 := NOT #FP_CMD.Start2 AND NOT #ONS.CMD_Start2;   // rising edge
   #ONS.CMD_Start2 := NOT #FP_CMD.Start2;
   #_w3 := NOT #FP_CMD.Start3 AND NOT #ONS.CMD_Start3;   // rising edge
   #ONS.CMD_Start3 := NOT #FP_CMD.Start3;
   #CMD_Stop := (#FP_CMD.Stop AND #FP_DIM.Stop) OR ((#_w1 OR #_w2 OR #_w3) AND #FP_SEL.INCH_Man AND #ModeManual);
END_REGION

REGION Network 57: Faceplate Commands Pulse Type - Stop
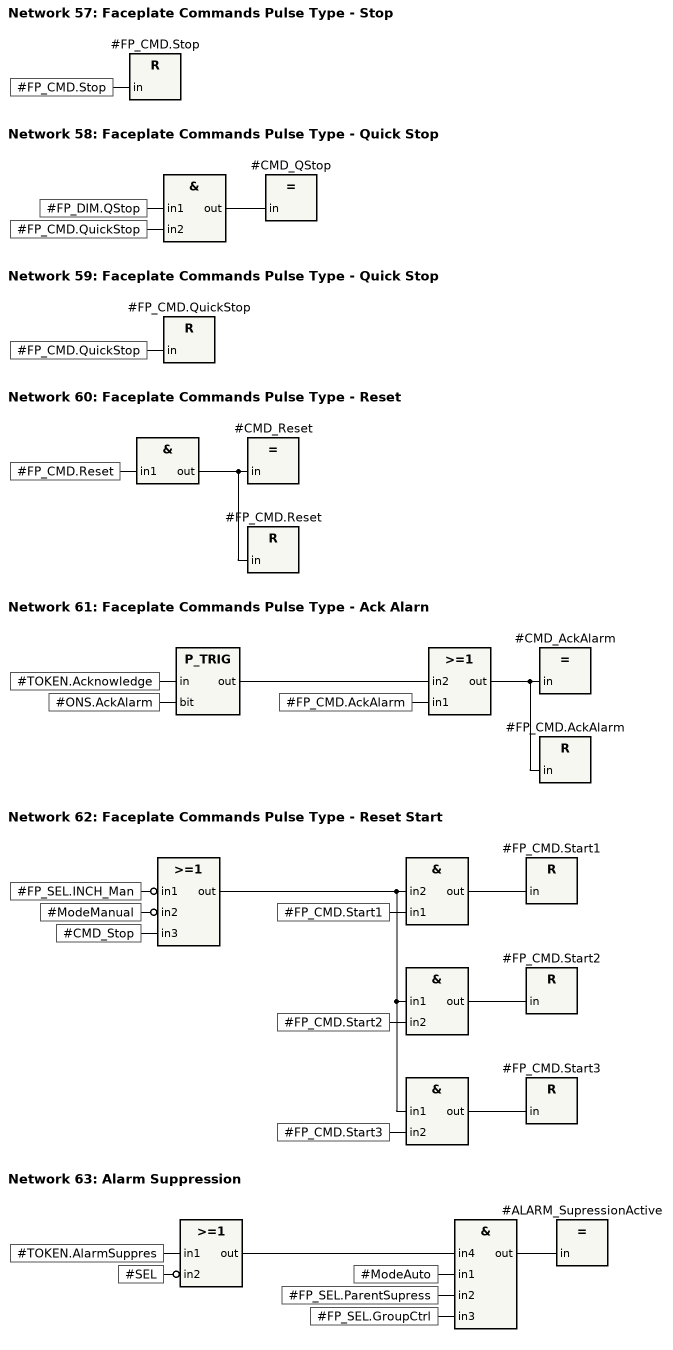
   IF #FP_CMD.Stop THEN #FP_CMD.Stop := FALSE; END_IF;
END_REGION

REGION Network 58: Faceplate Commands Pulse Type - Quick Stop
   #CMD_QStop := #FP_DIM.QStop AND #FP_CMD.QuickStop;
END_REGION

REGION Network 59: Faceplate Commands Pulse Type - Quick Stop
   IF #FP_CMD.QuickStop THEN #FP_CMD.QuickStop := FALSE; END_IF;
END_REGION

REGION Network 60: Faceplate Commands Pulse Type - Reset
   #CMD_Reset := #FP_CMD.Reset;
   IF #FP_CMD.Reset THEN #FP_CMD.Reset := FALSE; END_IF;
END_REGION

REGION Network 61: Faceplate Commands Pulse Type - Ack Alarn
   #_w1 := #TOKEN.Acknowledge AND NOT #ONS.AckAlarm;   // rising edge
   #ONS.AckAlarm := #TOKEN.Acknowledge;
   #CMD_AckAlarm := #_w1 OR #FP_CMD.AckAlarm;
   IF #CMD_AckAlarm THEN #FP_CMD.AckAlarm := FALSE; END_IF;
END_REGION

REGION Network 62: Faceplate Commands Pulse Type - Reset Start
   #_w1 := NOT #FP_SEL.INCH_Man OR NOT #ModeManual OR #CMD_Stop;
   IF #_w1 AND #FP_CMD.Start1 THEN #FP_CMD.Start1 := FALSE; END_IF;
   IF #_w1 AND #FP_CMD.Start2 THEN #FP_CMD.Start2 := FALSE; END_IF;
   IF #_w1 AND #FP_CMD.Start3 THEN #FP_CMD.Start3 := FALSE; END_IF;
END_REGION

REGION Network 63: Alarm Suppression
   #ALARM_SupressionActive := (#TOKEN.AlarmSuppres OR NOT #SEL) AND #ModeAuto AND #FP_SEL.ParentSupress AND #FP_SEL.GroupCtrl;
END_REGION

REGION Network 64: Child Alarm Suppression
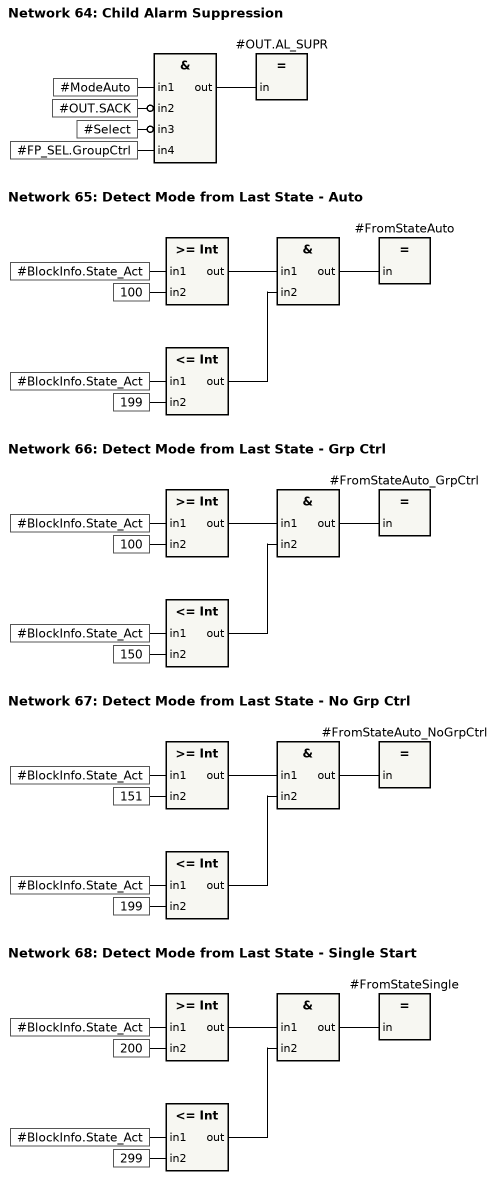
   #OUT.AL_SUPR := #ModeAuto AND NOT #OUT.SACK AND NOT #Select AND #FP_SEL.GroupCtrl;
END_REGION

REGION Network 65: Detect Mode from Last State - Auto
   #FromStateAuto := (#BlockInfo.State_Act >= 100) AND (#BlockInfo.State_Act <= 199);
END_REGION

REGION Network 66: Detect Mode from Last State - Grp Ctrl
   #FromStateAuto_GrpCtrl := (#BlockInfo.State_Act >= 100) AND (#BlockInfo.State_Act <= 150);
END_REGION

REGION Network 67: Detect Mode from Last State - No Grp Ctrl
   #FromStateAuto_NoGrpCtrl := (#BlockInfo.State_Act >= 151) AND (#BlockInfo.State_Act <= 199);
END_REGION

REGION Network 68: Detect Mode from Last State - Single Start
   #FromStateSingle := (#BlockInfo.State_Act >= 200) AND (#BlockInfo.State_Act <= 299);
END_REGION

REGION Network 69: Detect Mode from Last State - Manual
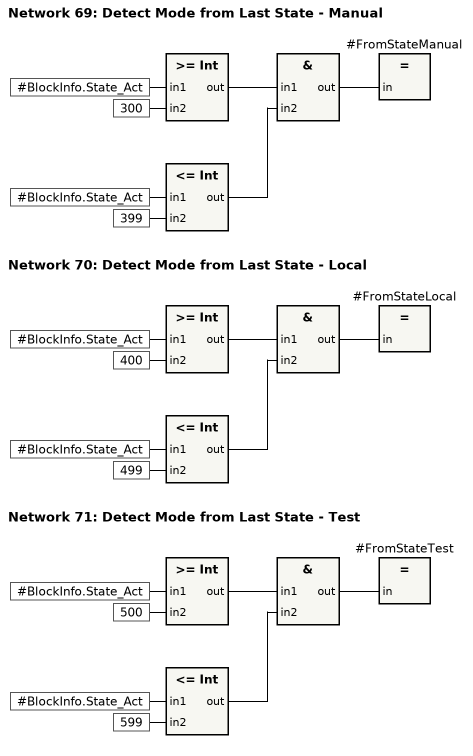
   #FromStateManual := (#BlockInfo.State_Act >= 300) AND (#BlockInfo.State_Act <= 399);
END_REGION

REGION Network 70: Detect Mode from Last State - Local
   #FromStateLocal := (#BlockInfo.State_Act >= 400) AND (#BlockInfo.State_Act <= 499);
END_REGION

REGION Network 71: Detect Mode from Last State - Test
   #FromStateTest := (#BlockInfo.State_Act >= 500) AND (#BlockInfo.State_Act <= 599);
END_REGION

REGION Network 72: Detect Mode from Last State
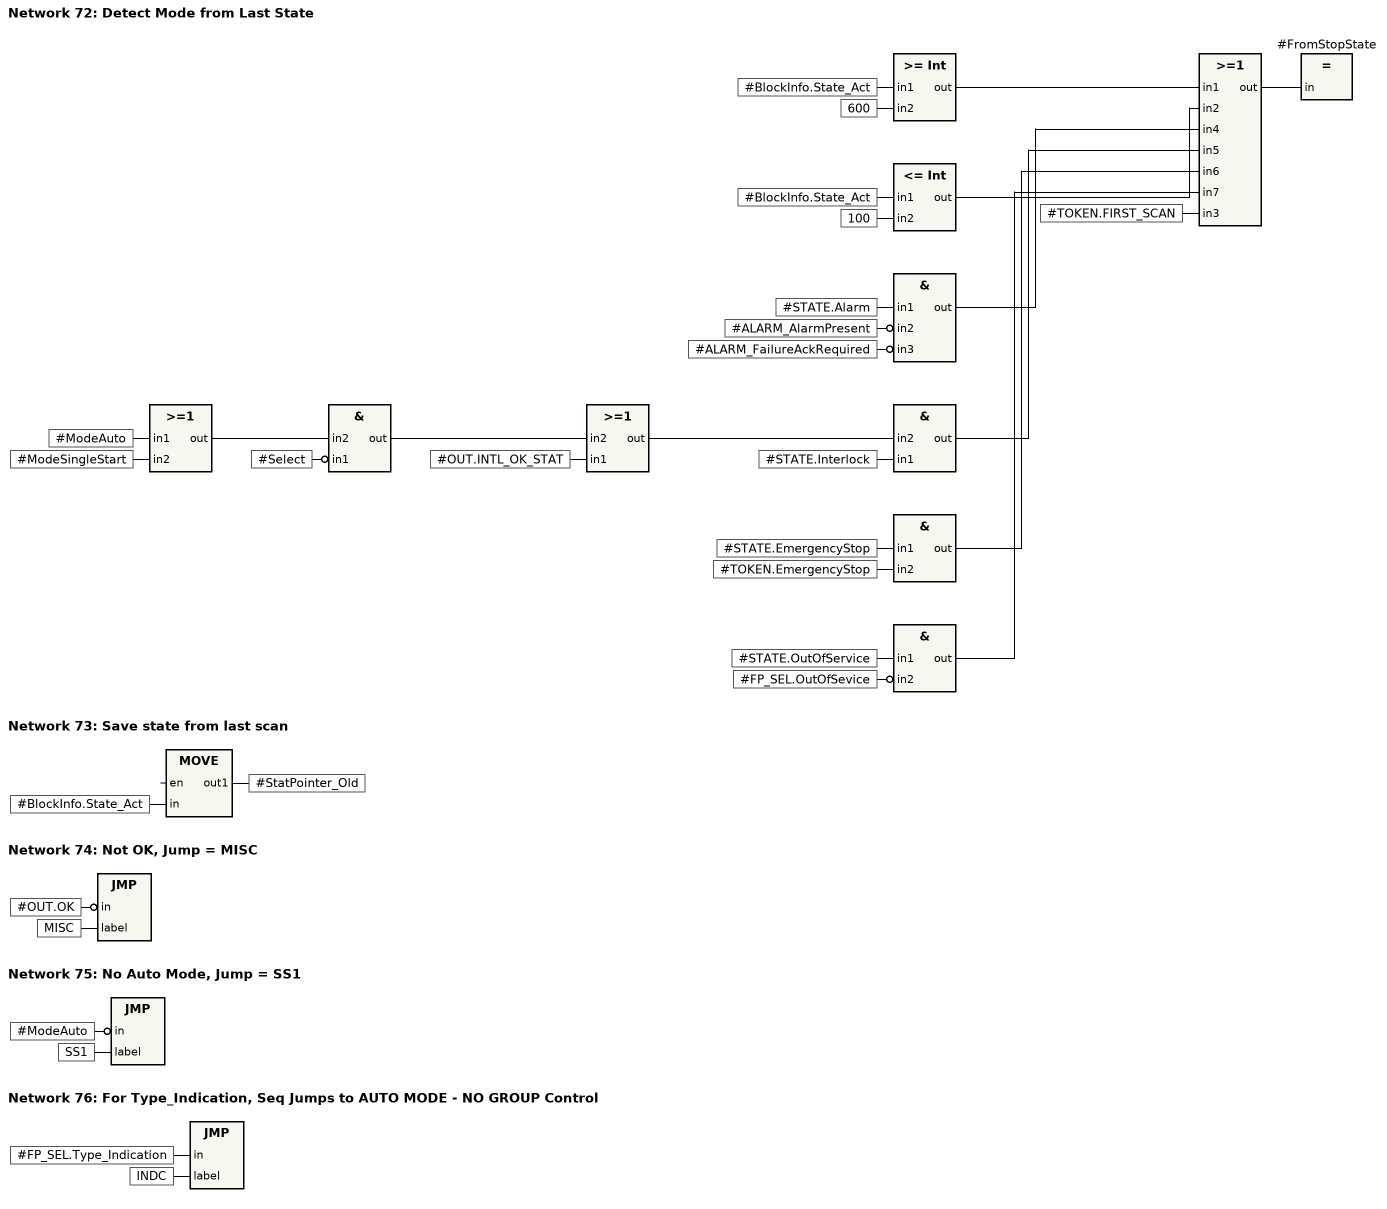
   #FromStopState := (#BlockInfo.State_Act >= 600) OR (#BlockInfo.State_Act <= 100) OR (#STATE.Alarm AND NOT #ALARM_AlarmPresent AND NOT #ALARM_FailureAckRequired) OR ((((#ModeAuto OR #ModeSingleStart) AND NOT #Select) OR #OUT.INTL_OK_STAT) AND #STATE.Interlock) OR (#STATE.EmergencyStop AND #TOKEN.EmergencyStop) OR (#STATE.OutOfService AND NOT #FP_SEL.OutOfSevice) OR #TOKEN.FIRST_SCAN;
END_REGION

REGION Network 73: Save state from last scan
   #StatPointer_Old := #BlockInfo.State_Act;
END_REGION

REGION Network 74: Not OK, Jump = MISC
   IF NOT #OUT.OK THEN GOTO MISC; END_IF;
END_REGION

REGION Network 75: No Auto Mode, Jump = SS1
   IF NOT #ModeAuto THEN GOTO SS1; END_IF;
END_REGION

REGION Network 76: For Type_Indication, Seq Jumps to AUTO MODE - NO GROUP Control
   IF #FP_SEL.Type_Indication THEN GOTO INDC; END_IF;
END_REGION

REGION Network 77: State: Auto - Stopped
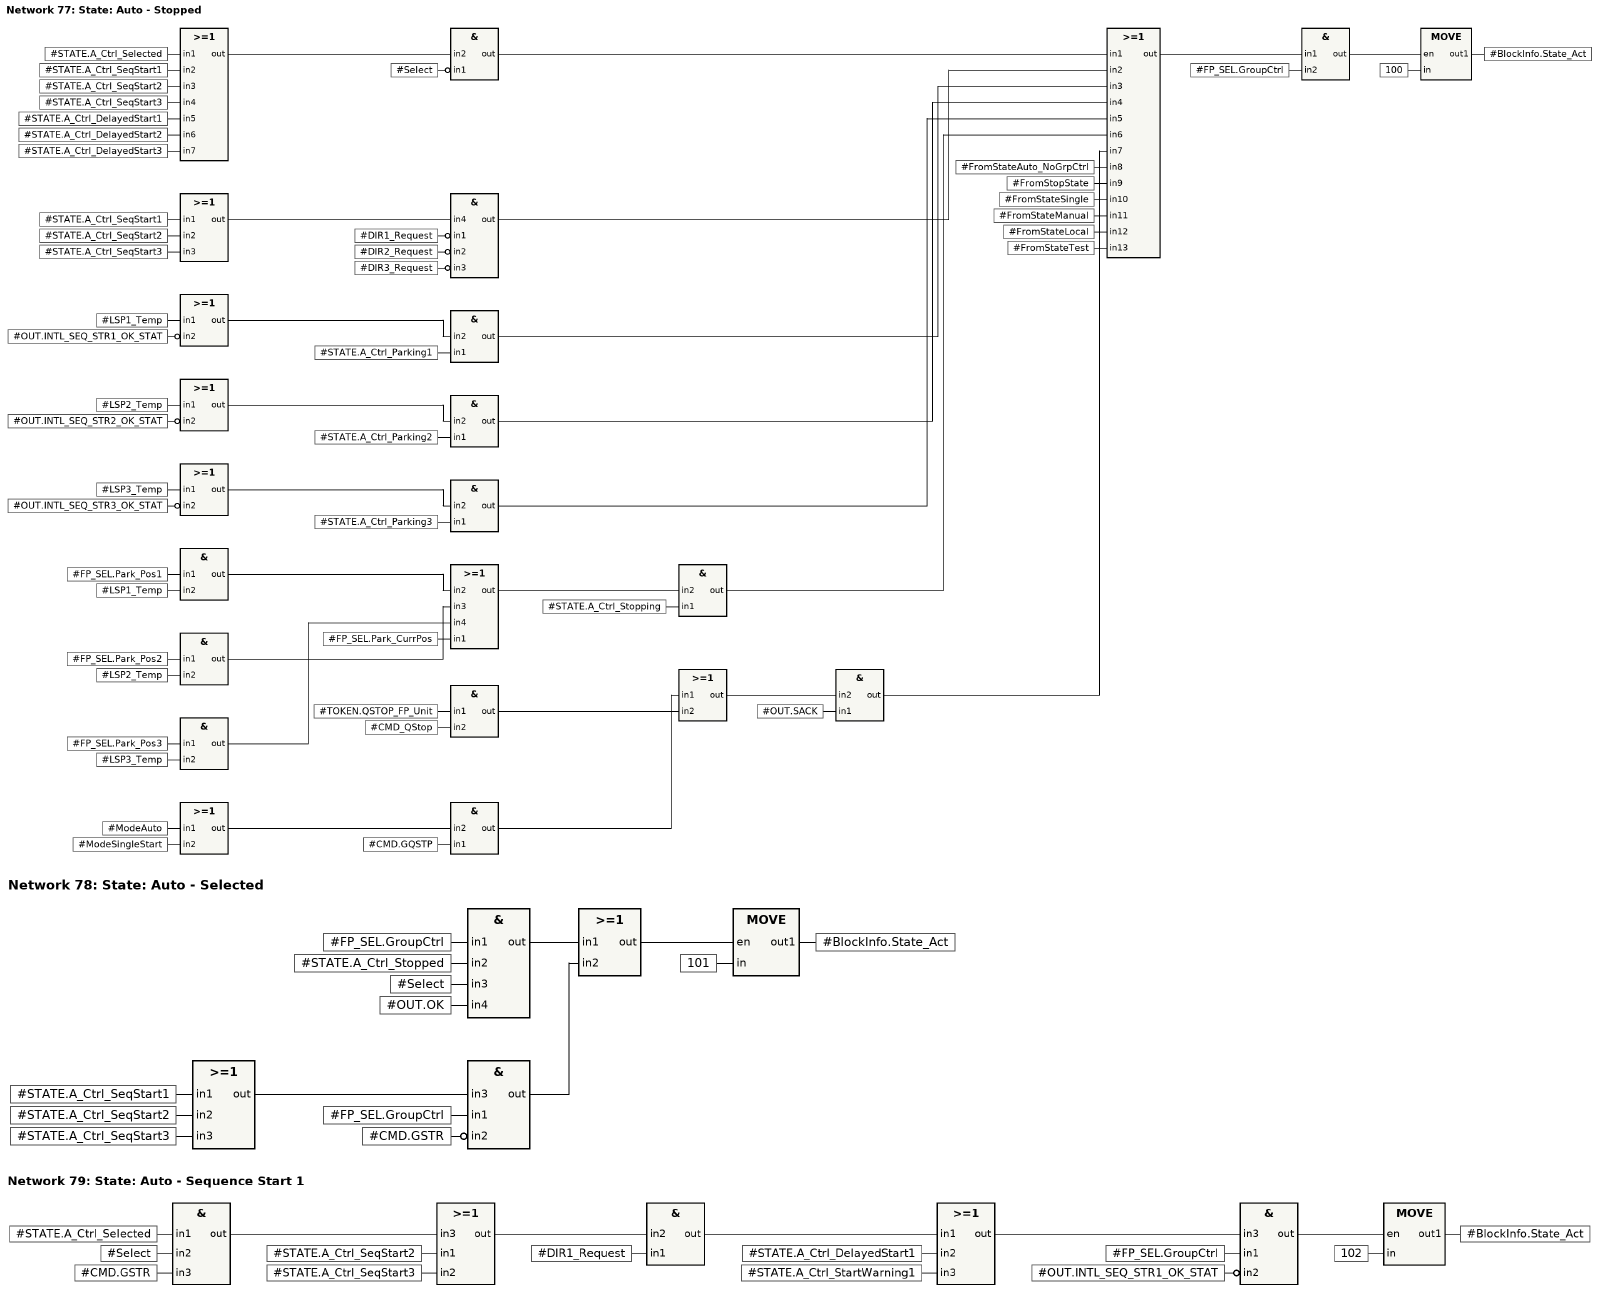
   IF (((#STATE.A_Ctrl_Selected OR #STATE.A_Ctrl_SeqStart1 OR #STATE.A_Ctrl_SeqStart2 OR #STATE.A_Ctrl_SeqStart3 OR #STATE.A_Ctrl_DelayedStart1 OR #STATE.A_Ctrl_DelayedStart2 OR #STATE.A_Ctrl_DelayedStart3) AND NOT #Select) OR ((#STATE.A_Ctrl_SeqStart1 OR #STATE.A_Ctrl_SeqStart2 OR #STATE.A_Ctrl_SeqStart3) AND NOT #DIR1_Request AND NOT #DIR2_Request AND NOT #DIR3_Request) OR ((#LSP1_Temp OR NOT #OUT.INTL_SEQ_STR1_OK_STAT) AND #STATE.A_Ctrl_Parking1) OR ((#LSP2_Temp OR NOT #OUT.INTL_SEQ_STR2_OK_STAT) AND #STATE.A_Ctrl_Parking2) OR ((#LSP3_Temp OR NOT #OUT.INTL_SEQ_STR3_OK_STAT) AND #STATE.A_Ctrl_Parking3) OR (((#FP_SEL.Park_Pos1 AND #LSP1_Temp) OR (#FP_SEL.Park_Pos2 AND #LSP2_Temp) OR (#FP_SEL.Park_Pos3 AND #LSP3_Temp) OR #FP_SEL.Park_CurrPos) AND #STATE.A_Ctrl_Stopping) OR ((((#ModeAuto OR #ModeSingleStart) AND #CMD.GQSTP) OR (#TOKEN.QSTOP_FP_Unit AND #CMD_QStop)) AND #OUT.SACK) OR #FromStateAuto_NoGrpCtrl OR #FromStopState OR #FromStateSingle OR #FromStateManual OR #FromStateLocal OR #FromStateTest) AND #FP_SEL.GroupCtrl THEN
       #BlockInfo.State_Act := 100;
   END_IF;
END_REGION

REGION Network 78: State: Auto - Selected
   IF (#FP_SEL.GroupCtrl AND #STATE.A_Ctrl_Stopped AND #Select AND #OUT.OK) OR ((#STATE.A_Ctrl_SeqStart1 OR #STATE.A_Ctrl_SeqStart2 OR #STATE.A_Ctrl_SeqStart3) AND #FP_SEL.GroupCtrl AND NOT #CMD.GSTR) THEN
       #BlockInfo.State_Act := 101;
   END_IF;
END_REGION

REGION Network 79: State: Auto - Sequence Start 1
   IF ((((#STATE.A_Ctrl_Selected AND #Select AND #CMD.GSTR) OR #STATE.A_Ctrl_SeqStart2 OR #STATE.A_Ctrl_SeqStart3) AND #DIR1_Request) OR #STATE.A_Ctrl_DelayedStart1 OR #STATE.A_Ctrl_StartWarning1) AND #FP_SEL.GroupCtrl AND NOT #OUT.INTL_SEQ_STR1_OK_STAT THEN
       #BlockInfo.State_Act := 102;
   END_IF;
END_REGION

REGION Network 80: State: Auto - Sequence Start 2
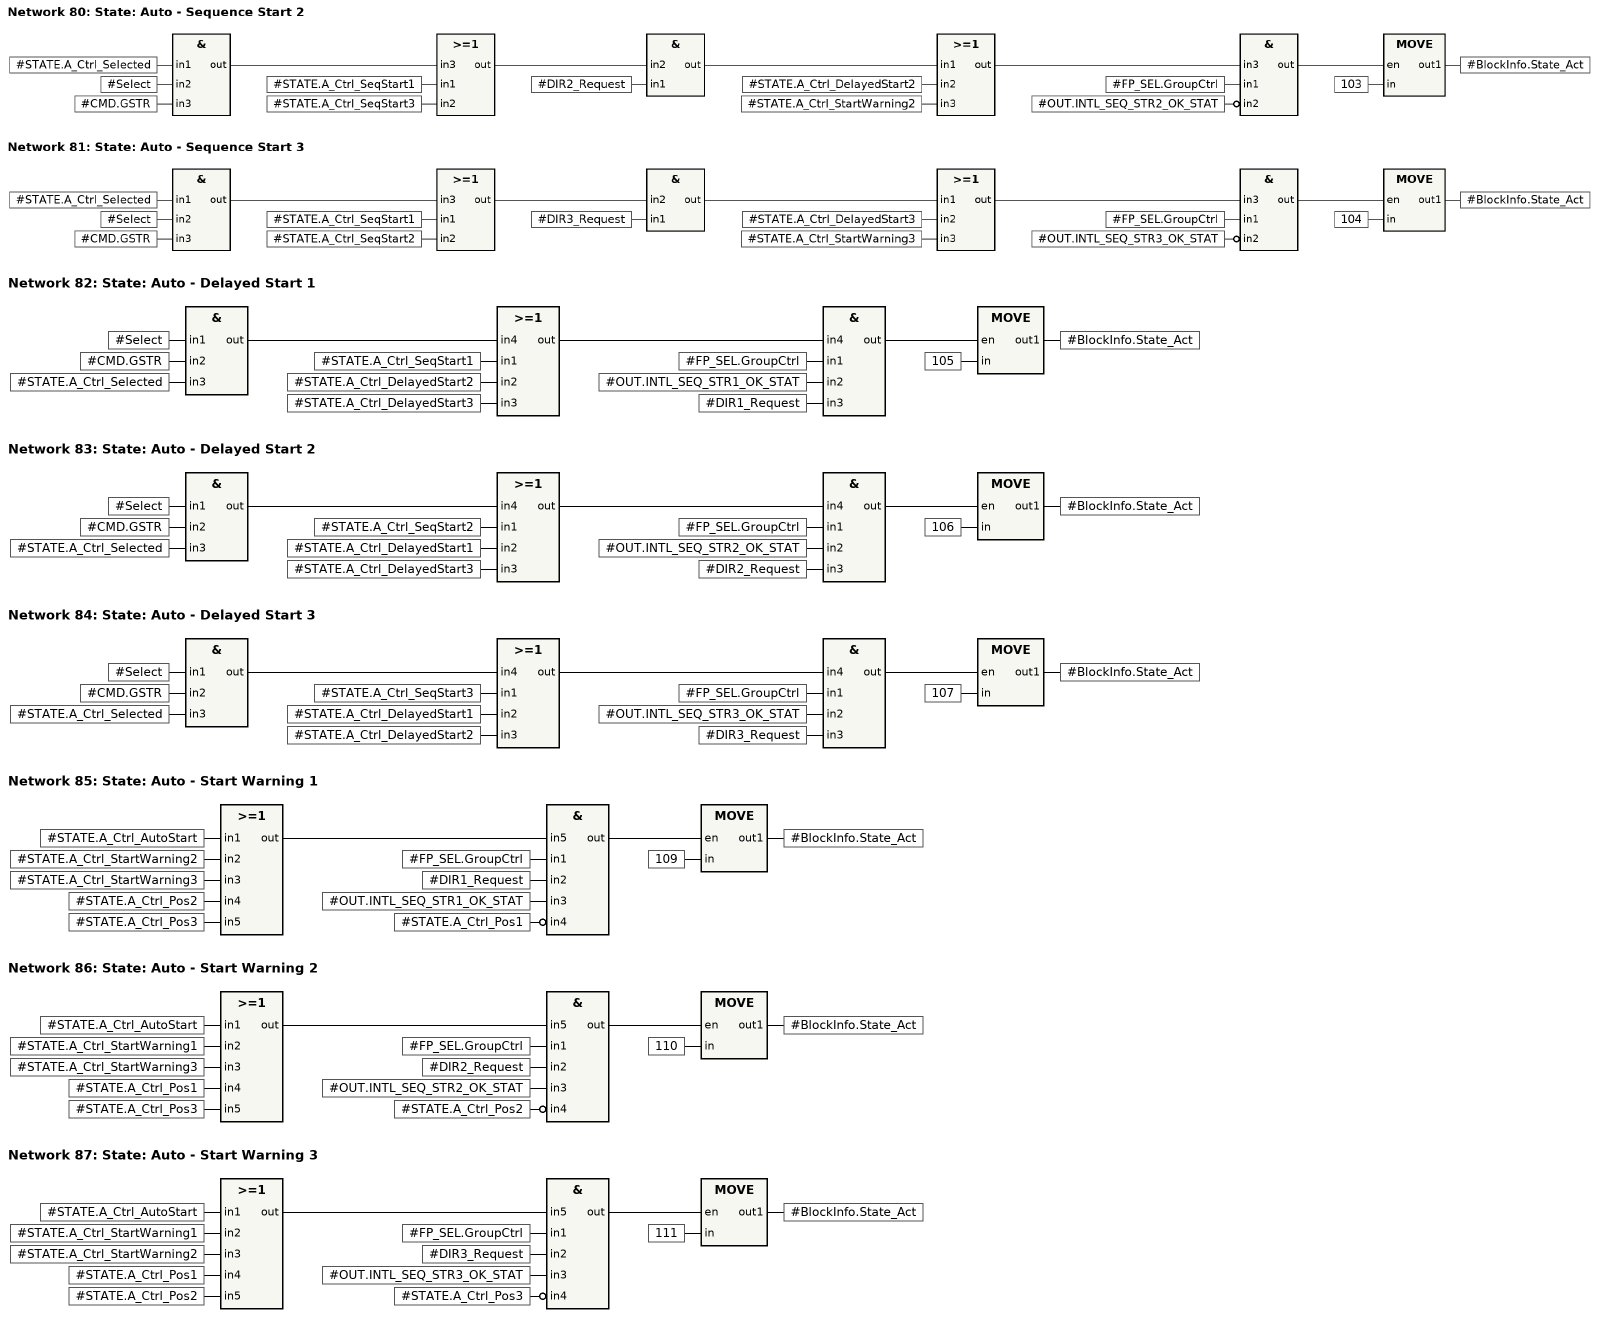
   IF ((((#STATE.A_Ctrl_Selected AND #Select AND #CMD.GSTR) OR #STATE.A_Ctrl_SeqStart1 OR #STATE.A_Ctrl_SeqStart3) AND #DIR2_Request) OR #STATE.A_Ctrl_DelayedStart2 OR #STATE.A_Ctrl_StartWarning2) AND #FP_SEL.GroupCtrl AND NOT #OUT.INTL_SEQ_STR2_OK_STAT THEN
       #BlockInfo.State_Act := 103;
   END_IF;
END_REGION

REGION Network 81: State: Auto - Sequence Start 3
   IF ((((#STATE.A_Ctrl_Selected AND #Select AND #CMD.GSTR) OR #STATE.A_Ctrl_SeqStart1 OR #STATE.A_Ctrl_SeqStart2) AND #DIR3_Request) OR #STATE.A_Ctrl_DelayedStart3 OR #STATE.A_Ctrl_StartWarning3) AND #FP_SEL.GroupCtrl AND NOT #OUT.INTL_SEQ_STR3_OK_STAT THEN
       #BlockInfo.State_Act := 104;
   END_IF;
END_REGION

REGION Network 82: State: Auto - Delayed Start 1
   IF ((#Select AND #CMD.GSTR AND #STATE.A_Ctrl_Selected) OR #STATE.A_Ctrl_SeqStart1 OR #STATE.A_Ctrl_DelayedStart2 OR #STATE.A_Ctrl_DelayedStart3) AND #FP_SEL.GroupCtrl AND #OUT.INTL_SEQ_STR1_OK_STAT AND #DIR1_Request THEN
       #BlockInfo.State_Act := 105;
   END_IF;
END_REGION

REGION Network 83: State: Auto - Delayed Start 2
   IF ((#Select AND #CMD.GSTR AND #STATE.A_Ctrl_Selected) OR #STATE.A_Ctrl_SeqStart2 OR #STATE.A_Ctrl_DelayedStart1 OR #STATE.A_Ctrl_DelayedStart3) AND #FP_SEL.GroupCtrl AND #OUT.INTL_SEQ_STR2_OK_STAT AND #DIR2_Request THEN
       #BlockInfo.State_Act := 106;
   END_IF;
END_REGION

REGION Network 84: State: Auto - Delayed Start 3
   IF ((#Select AND #CMD.GSTR AND #STATE.A_Ctrl_Selected) OR #STATE.A_Ctrl_SeqStart3 OR #STATE.A_Ctrl_DelayedStart1 OR #STATE.A_Ctrl_DelayedStart2) AND #FP_SEL.GroupCtrl AND #OUT.INTL_SEQ_STR3_OK_STAT AND #DIR3_Request THEN
       #BlockInfo.State_Act := 107;
   END_IF;
END_REGION

REGION Network 85: State: Auto - Start Warning 1
   IF (#STATE.A_Ctrl_AutoStart OR #STATE.A_Ctrl_StartWarning2 OR #STATE.A_Ctrl_StartWarning3 OR #STATE.A_Ctrl_Pos2 OR #STATE.A_Ctrl_Pos3) AND #FP_SEL.GroupCtrl AND #DIR1_Request AND #OUT.INTL_SEQ_STR1_OK_STAT AND NOT #STATE.A_Ctrl_Pos1 THEN
       #BlockInfo.State_Act := 109;
   END_IF;
END_REGION

REGION Network 86: State: Auto - Start Warning 2
   IF (#STATE.A_Ctrl_AutoStart OR #STATE.A_Ctrl_StartWarning1 OR #STATE.A_Ctrl_StartWarning3 OR #STATE.A_Ctrl_Pos1 OR #STATE.A_Ctrl_Pos3) AND #FP_SEL.GroupCtrl AND #DIR2_Request AND #OUT.INTL_SEQ_STR2_OK_STAT AND NOT #STATE.A_Ctrl_Pos2 THEN
       #BlockInfo.State_Act := 110;
   END_IF;
END_REGION

REGION Network 87: State: Auto - Start Warning 3
   IF (#STATE.A_Ctrl_AutoStart OR #STATE.A_Ctrl_StartWarning1 OR #STATE.A_Ctrl_StartWarning2 OR #STATE.A_Ctrl_Pos1 OR #STATE.A_Ctrl_Pos2) AND #FP_SEL.GroupCtrl AND #DIR3_Request AND #OUT.INTL_SEQ_STR3_OK_STAT AND NOT #STATE.A_Ctrl_Pos3 THEN
       #BlockInfo.State_Act := 111;
   END_IF;
END_REGION

REGION Network 88: State: Auto - Running 1
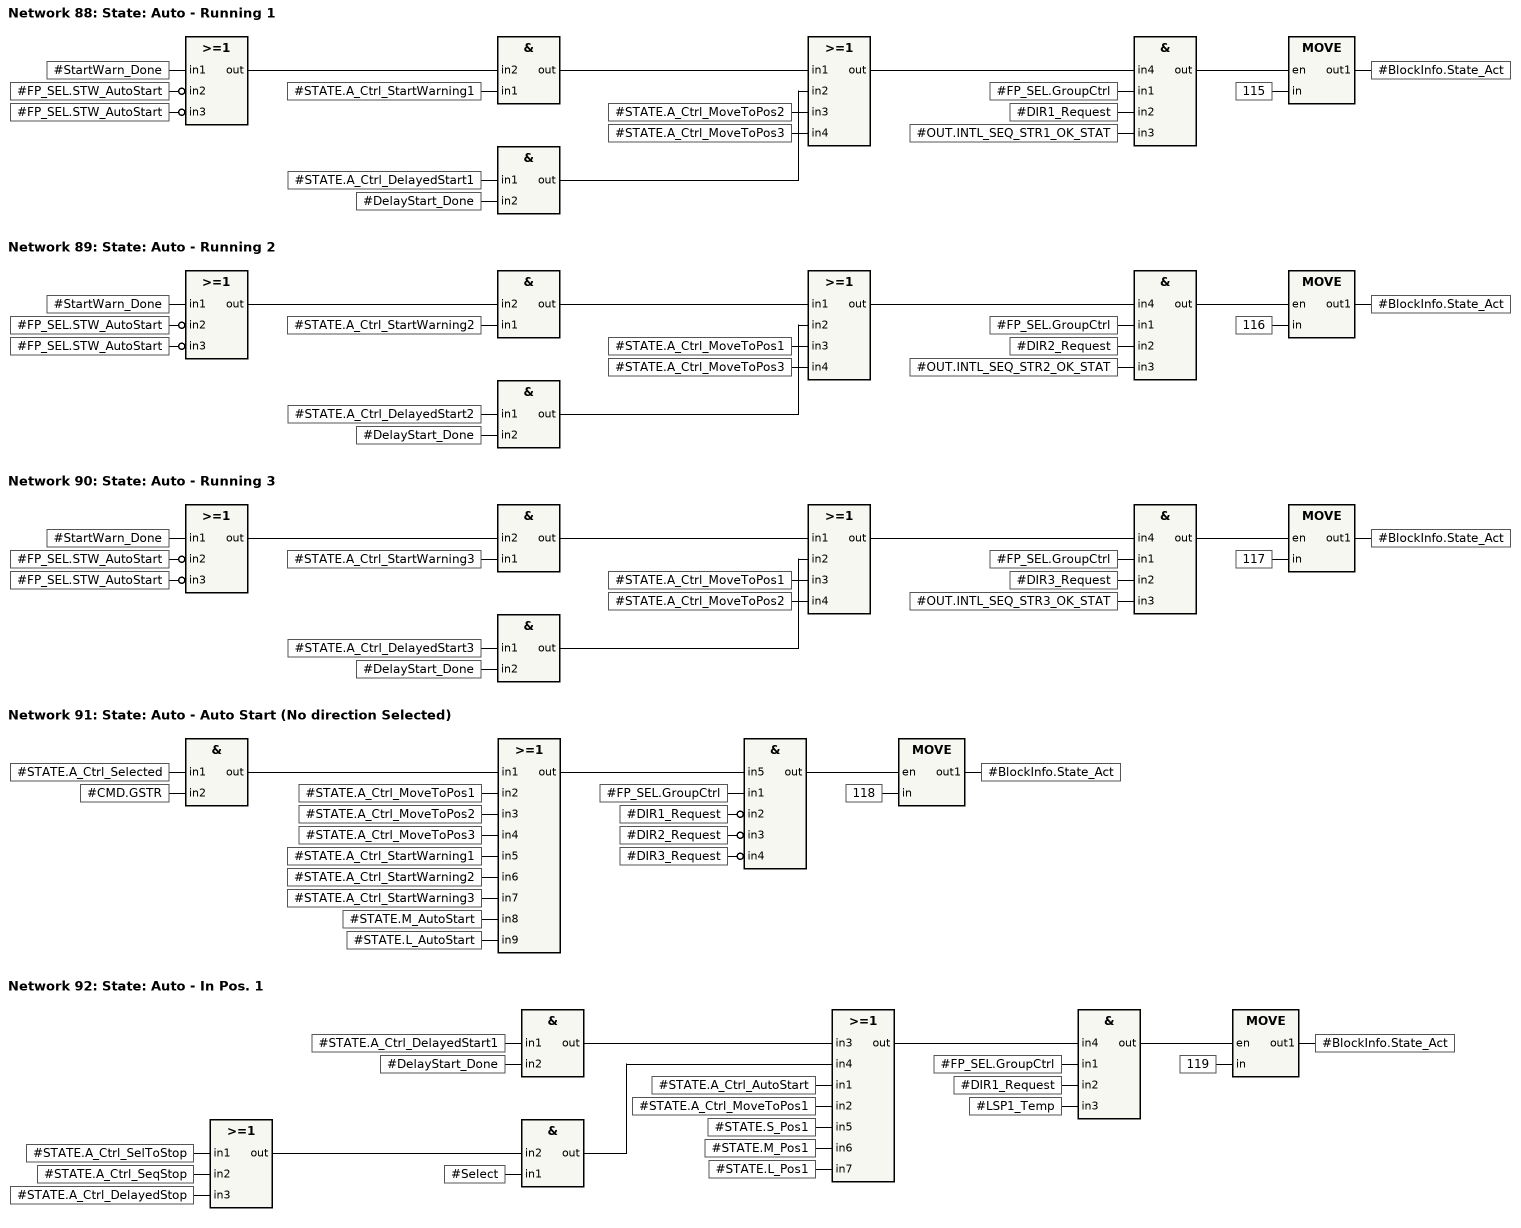
   IF (((#StartWarn_Done OR NOT #FP_SEL.STW_AutoStart OR NOT #FP_SEL.STW_AutoStart) AND #STATE.A_Ctrl_StartWarning1) OR (#STATE.A_Ctrl_DelayedStart1 AND #DelayStart_Done) OR #STATE.A_Ctrl_MoveToPos2 OR #STATE.A_Ctrl_MoveToPos3) AND #FP_SEL.GroupCtrl AND #DIR1_Request AND #OUT.INTL_SEQ_STR1_OK_STAT THEN
       #BlockInfo.State_Act := 115;
   END_IF;
END_REGION

REGION Network 89: State: Auto - Running 2
   IF (((#StartWarn_Done OR NOT #FP_SEL.STW_AutoStart OR NOT #FP_SEL.STW_AutoStart) AND #STATE.A_Ctrl_StartWarning2) OR (#STATE.A_Ctrl_DelayedStart2 AND #DelayStart_Done) OR #STATE.A_Ctrl_MoveToPos1 OR #STATE.A_Ctrl_MoveToPos3) AND #FP_SEL.GroupCtrl AND #DIR2_Request AND #OUT.INTL_SEQ_STR2_OK_STAT THEN
       #BlockInfo.State_Act := 116;
   END_IF;
END_REGION

REGION Network 90: State: Auto - Running 3
   IF (((#StartWarn_Done OR NOT #FP_SEL.STW_AutoStart OR NOT #FP_SEL.STW_AutoStart) AND #STATE.A_Ctrl_StartWarning3) OR (#STATE.A_Ctrl_DelayedStart3 AND #DelayStart_Done) OR #STATE.A_Ctrl_MoveToPos1 OR #STATE.A_Ctrl_MoveToPos2) AND #FP_SEL.GroupCtrl AND #DIR3_Request AND #OUT.INTL_SEQ_STR3_OK_STAT THEN
       #BlockInfo.State_Act := 117;
   END_IF;
END_REGION

REGION Network 91: State: Auto - Auto Start (No direction Selected)
   IF ((#STATE.A_Ctrl_Selected AND #CMD.GSTR) OR #STATE.A_Ctrl_MoveToPos1 OR #STATE.A_Ctrl_MoveToPos2 OR #STATE.A_Ctrl_MoveToPos3 OR #STATE.A_Ctrl_StartWarning1 OR #STATE.A_Ctrl_StartWarning2 OR #STATE.A_Ctrl_StartWarning3 OR #STATE.M_AutoStart OR #STATE.L_AutoStart) AND #FP_SEL.GroupCtrl AND NOT #DIR1_Request AND NOT #DIR2_Request AND NOT #DIR3_Request THEN
       #BlockInfo.State_Act := 118;
   END_IF;
END_REGION

REGION Network 92: State: Auto - In Pos. 1
   IF ((#STATE.A_Ctrl_DelayedStart1 AND #DelayStart_Done) OR ((#STATE.A_Ctrl_SelToStop OR #STATE.A_Ctrl_SeqStop OR #STATE.A_Ctrl_DelayedStop) AND #Select) OR #STATE.A_Ctrl_AutoStart OR #STATE.A_Ctrl_MoveToPos1 OR #STATE.S_Pos1 OR #STATE.M_Pos1 OR #STATE.L_Pos1) AND #FP_SEL.GroupCtrl AND #DIR1_Request AND #LSP1_Temp THEN
       #BlockInfo.State_Act := 119;
   END_IF;
END_REGION

REGION Network 93: State: Auto - In Pos. 2
